# B&R Automation Studio project AAU12Segmenter (part 7)

#### DemoProgram.st - not listed in the package file held
```iecst
ACTION demoProgramTask:
	positionContainerDemo_0[0].initXPos := 0.060;
	positionContainerDemo_0[0].initYPos := 0.120;
	positionContainerDemo_0[1].initXPos := 0.180;
	positionContainerDemo_0[1].initYPos := 0.120;
	positionContainerDemo_0[2].initXPos := 0.300;
	positionContainerDemo_0[2].initYPos := 0.120;
	positionContainerDemo_0[3].initXPos := 0.420;
	positionContainerDemo_0[3].initYPos := 0.120;

	//Setup
	positionContainerLinkMovement[0].Shuttle3.xPos := 0.120;
	positionContainerLinkMovement[0].Shuttle3.yPos := 0.120;
	positionContainerLinkMovement[0].Shuttle2.xPos := 0.360;
	positionContainerLinkMovement[0].Shuttle2.yPos := 0.360;
	positionContainerLinkMovement[0].Shuttle4.xPos := 0.360;
	positionContainerLinkMovement[0].Shuttle4.yPos := 0.120;
	positionContainerLinkMovement[0].Shuttle1.xPos := 0.120;
	positionContainerLinkMovement[0].Shuttle1.yPos := 0.360;

	positionContainerLinkMovement[1].Shuttle3.xPos := 0.060;
	positionContainerLinkMovement[1].Shuttle3.yPos := 0.060;
	positionContainerLinkMovement[1].Shuttle2.xPos := 0.180;
	positionContainerLinkMovement[1].Shuttle2.yPos := 0.180;
	positionContainerLinkMovement[1].Shuttle4.xPos := 0.180;
	positionContainerLinkMovement[1].Shuttle4.yPos := 0.060;
	positionContainerLinkMovement[1].Shuttle1.xPos := 0.060;
	positionContainerLinkMovement[1].Shuttle1.yPos := 0.180;

	positionContainerLinkMovement[2].Shuttle3.xPos := 0.120;
	positionContainerLinkMovement[2].Shuttle3.yPos := 0.120;
	positionContainerLinkMovement[2].Shuttle2.xPos := 0.360;
	positionContainerLinkMovement[2].Shuttle2.yPos := 0.360;
	positionContainerLinkMovement[2].Shuttle4.xPos := 0.360;
	positionContainerLinkMovement[2].Shuttle4.yPos := 0.120;
	positionContainerLinkMovement[2].Shuttle1.xPos := 0.120;
	positionContainerLinkMovement[2].Shuttle1.yPos := 0.360;

	positionContainerLinkMovement[3].Shuttle3.xPos := 0.300;
	positionContainerLinkMovement[3].Shuttle3.yPos := 0.060;
	positionContainerLinkMovement[3].Shuttle2.xPos := 0.420;
	positionContainerLinkMovement[3].Shuttle2.yPos := 0.180;
	positionContainerLinkMovement[3].Shuttle4.xPos := 0.420;
	positionContainerLinkMovement[3].Shuttle4.yPos := 0.060;
	positionContainerLinkMovement[3].Shuttle1.xPos := 0.300;
	positionContainerLinkMovement[3].Shuttle1.yPos := 0.180;

	positionContainerLinkMovement[4].Shuttle3.xPos := 0.120;
	positionContainerLinkMovement[4].Shuttle3.yPos := 0.120;
	positionContainerLinkMovement[4].Shuttle2.xPos := 0.360;
	positionContainerLinkMovement[4].Shuttle2.yPos := 0.360;
	positionContainerLinkMovement[4].Shuttle4.xPos := 0.360;
	positionContainerLinkMovement[4].Shuttle4.yPos := 0.120;
	positionContainerLinkMovement[4].Shuttle1.xPos := 0.120;
	positionContainerLinkMovement[4].Shuttle1.yPos := 0.360;

	positionContainerLinkMovement[5].Shuttle3.xPos := 0.300;
	positionContainerLinkMovement[5].Shuttle3.yPos := 0.300;
	positionContainerLinkMovement[5].Shuttle2.xPos := 0.420;
	positionContainerLinkMovement[5].Shuttle2.yPos := 0.420;
	positionContainerLinkMovement[5].Shuttle4.xPos := 0.420;
	positionContainerLinkMovement[5].Shuttle4.yPos := 0.300;
	positionContainerLinkMovement[5].Shuttle1.xPos := 0.300;
	positionContainerLinkMovement[5].Shuttle1.yPos := 0.420;

	positionContainerLinkMovement[6].Shuttle3.xPos := 0.120;
	positionContainerLinkMovement[6].Shuttle3.yPos := 0.120;
	positionContainerLinkMovement[6].Shuttle2.xPos := 0.360;
	positionContainerLinkMovement[6].Shuttle2.yPos := 0.360;
	positionContainerLinkMovement[6].Shuttle4.xPos := 0.360;
	positionContainerLinkMovement[6].Shuttle4.yPos := 0.120;
	positionContainerLinkMovement[6].Shuttle1.xPos := 0.120;
	positionContainerLinkMovement[6].Shuttle1.yPos := 0.360;

	CASE em.substate OF
		5000:

			em.description := 'Move shuttle to pre pos';
			tempShuttleCounter := 0;
			MC_BR_MoveInPlaneAsync_Acp6D_0.Parameters.Acceleration := gAcp6DCtrl.Par.Acceleration;
			MC_BR_MoveInPlaneAsync_Acp6D_0.Parameters.Velocity := gAcp6DCtrl.Par.Velocity;
			FOR i := 0 TO UINT_TO_USINT(localCurrentNumShuttles-1) DO
				MC_BR_MoveInPlaneAsync_Acp6D_0.Parameters.AsyncPar[i].Shuttle := ADR(gAcp6DCtrl.Status.ShuttleInfo[i].shuttleRef);
				MC_BR_MoveInPlaneAsync_Acp6D_0.Parameters.AsyncPar[i].X := positionContainerDemo_0[i].initXPos;
				MC_BR_MoveInPlaneAsync_Acp6D_0.Parameters.AsyncPar[i].Y := positionContainerDemo_0[i].initYPos;
			END_FOR
			MC_BR_MoveInPlaneAsync_Acp6D_0.Execute := TRUE;
			IF MC_BR_MoveInPlaneAsync_Acp6D_0.Acknowledge THEN
				MC_BR_MoveInPlaneAsync_Acp6D_0.Execute := FALSE;
				em.substate := 5010;
			END_IF

		5010:
			MC_BR_MacroRun_Acp6D_0.Name := 'shuttleWave';
			MC_BR_MacroRun_Acp6D_0.Shuttle := ADR(gAcp6DCtrl.Status.ShuttleInfo[0].shuttleRef);
			MC_BR_MacroRun_Acp6D_0.Execute := TRUE;
			IF MC_BR_MacroRun_Acp6D_0.Acknowledge THEN
				MC_BR_MacroRun_Acp6D_0.Execute := FALSE;
				em.substate := 5015;
			END_IF

		5015:
			TON_0.PT := t#500ms;
			TON_0.IN := TRUE;
			IF TON_0.Q THEN
				TON_0.IN := FALSE;
				em.substate := 5020;
			END_IF

		5020:
			MC_BR_MacroRun_Acp6D_0.Name := 'shuttleWave';
			MC_BR_MacroRun_Acp6D_0.Shuttle := ADR(gAcp6DCtrl.Status.ShuttleInfo[1].shuttleRef);
			MC_BR_MacroRun_Acp6D_0.Execute := TRUE;
			IF MC_BR_MacroRun_Acp6D_0.Acknowledge THEN
				MC_BR_MacroRun_Acp6D_0.Execute := FALSE;
				em.substate := 5025;
			END_IF

		5025:
			TON_0.PT := t#500ms;
			TON_0.IN := TRUE;
			IF TON_0.Q THEN
				TON_0.IN := FALSE;
				em.substate := 5030;
			END_IF

		5030:
			MC_BR_MacroRun_Acp6D_0.Name := 'shuttleWave';
			MC_BR_MacroRun_Acp6D_0.Shuttle := ADR(gAcp6DCtrl.Status.ShuttleInfo[2].shuttleRef);
			MC_BR_MacroRun_Acp6D_0.Execute := TRUE;
			IF MC_BR_MacroRun_Acp6D_0.Acknowledge THEN
				MC_BR_MacroRun_Acp6D_0.Execute := FALSE;
				em.substate := 5035;
			END_IF

		5035:
			TON_0.PT := t#500ms;
			TON_0.IN := TRUE;
			IF TON_0.Q THEN
				TON_0.IN := FALSE;
				em.substate := 5040;
			END_IF

		5040:
			MC_BR_MacroRun_Acp6D_0.Name := 'shuttleWave';
			MC_BR_MacroRun_Acp6D_0.Shuttle := ADR(gAcp6DCtrl.Status.ShuttleInfo[3].shuttleRef);
			MC_BR_MacroRun_Acp6D_0.Execute := TRUE;
			IF MC_BR_MacroRun_Acp6D_0.Acknowledge THEN
				MC_BR_MacroRun_Acp6D_0.Execute := FALSE;
				em.substate := 5045;
			END_IF

		5045:
			em.description := 'Check all shuttle state';
			IF gAcp6DCtrl.Status.ShuttleInfo[0].State = mcACP6D_SH_STATE_IDLING AND gAcp6DCtrl.Status.ShuttleInfo[1].State = mcACP6D_SH_STATE_IDLING
				AND gAcp6DCtrl.Status.ShuttleInfo[2].State = mcACP6D_SH_STATE_IDLING AND gAcp6DCtrl.Status.ShuttleInfo[3].State = mcACP6D_SH_STATE_IDLING AND MC_BR_AsmReadStatus_Acp6D_0.AssemblyReady THEN
				em.substate := 5050;
			END_IF

		5050:
			em.description := 'Couple ShuttleGroup1_2';
			em.cmd.sc := FALSE;
			MC_BR_ShGroupCoupleCtrl_Acp6D_0.ShuttleGroup := shGroupShuttle1_2;
			MC_BR_ShGroupCoupleCtrl_Acp6D_0.Parameters.Option := 1; //Couple
			MC_BR_ShGroupCoupleCtrl_Acp6D_0.Execute := TRUE;
			IF MC_BR_ShGroupCoupleCtrl_Acp6D_0.Done THEN
				MC_BR_ShGroupCoupleCtrl_Acp6D_0.Execute := FALSE;
				em.substate := 5060;
			END_IF

		5060:
			em.description := 'Couple ShuttleGroup3_4';
			em.cmd.sc := FALSE;
			MC_BR_ShGroupCoupleCtrl_Acp6D_0.ShuttleGroup := shGroupShuttle3_4;
			MC_BR_ShGroupCoupleCtrl_Acp6D_0.Parameters.Option := 1; //Couple
			MC_BR_ShGroupCoupleCtrl_Acp6D_0.Execute := TRUE;
			IF MC_BR_ShGroupCoupleCtrl_Acp6D_0.Done THEN
				MC_BR_ShGroupCoupleCtrl_Acp6D_0.Execute := FALSE;
				em.substate := 5070;
			END_IF

		5070:
			em.cmd.sc := FALSE;
			MC_BR_MoveInPlane_Acp6D_0.Shuttle := ADR(gAcp6DCtrl.Status.ShuttleInfo[0].shuttleRef);
			MC_BR_MoveInPlane_Acp6D_0.Parameters.Position.X := 0.060;
			MC_BR_MoveInPlane_Acp6D_0.Parameters.Position.Y := 0.060;
			MC_BR_MoveInPlane_Acp6D_0.Parameters.Velocity := gAcp6DCtrl.Par.Velocity;
			MC_BR_MoveInPlane_Acp6D_0.Parameters.Acceleration := gAcp6DCtrl.Par.Acceleration;
			MC_BR_MoveInPlane_Acp6D_0.Parameters.Mode := 0; //Abs
			MC_BR_MoveInPlane_Acp6D_0.Parameters.Path := 0; //direct
			MC_BR_MoveInPlane_Acp6D_0.Execute := TRUE;
			IF MC_BR_MoveInPlane_Acp6D_0.Acknowledge THEN
				MC_BR_MoveInPlane_Acp6D_0.Execute := FALSE;
				em.substate := 5080;
			END_IF

		5080:
			em.cmd.sc := FALSE;
			MC_BR_MoveInPlane_Acp6D_0.Shuttle := ADR(gAcp6DCtrl.Status.ShuttleInfo[0].shuttleRef);
			MC_BR_MoveInPlane_Acp6D_0.Parameters.Position.X := 0.300;
			MC_BR_MoveInPlane_Acp6D_0.Parameters.Position.Y := 0.060;
			MC_BR_MoveInPlane_Acp6D_0.Parameters.Velocity := gAcp6DCtrl.Par.Velocity;
			MC_BR_MoveInPlane_Acp6D_0.Parameters.Acceleration := gAcp6DCtrl.Par.Acceleration;
			MC_BR_MoveInPlane_Acp6D_0.Parameters.Mode := 0; //Abs
			MC_BR_MoveInPlane_Acp6D_0.Parameters.Path := 0; //direct
			MC_BR_MoveInPlane_Acp6D_0.Execute := TRUE;
			IF MC_BR_MoveInPlane_Acp6D_0.Acknowledge THEN
				MC_BR_MoveInPlane_Acp6D_0.Execute := FALSE;
				em.substate := 5090;
			END_IF

		5090:
			em.cmd.sc := FALSE;
			MC_BR_MoveInPlane_Acp6D_0.Shuttle := ADR(gAcp6DCtrl.Status.ShuttleInfo[0].shuttleRef);
			MC_BR_MoveInPlane_Acp6D_0.Parameters.Position.X := 0.060;
			MC_BR_MoveInPlane_Acp6D_0.Parameters.Position.Y := 0.060;
			MC_BR_MoveInPlane_Acp6D_0.Parameters.Velocity := gAcp6DCtrl.Par.Velocity;
			MC_BR_MoveInPlane_Acp6D_0.Parameters.Acceleration := gAcp6DCtrl.Par.Acceleration;
			MC_BR_MoveInPlane_Acp6D_0.Parameters.Mode := 0; //Abs
			MC_BR_MoveInPlane_Acp6D_0.Parameters.Path := 0; //direct
			MC_BR_MoveInPlane_Acp6D_0.Execute := TRUE;
			IF MC_BR_MoveInPlane_Acp6D_0.Acknowledge THEN
				MC_BR_MoveInPlane_Acp6D_0.Execute := FALSE;
				em.substate := 5100;
			END_IF

		5100:
			em.cmd.sc := FALSE;
			MC_BR_MoveInPlane_Acp6D_0.Shuttle := ADR(gAcp6DCtrl.Status.ShuttleInfo[0].shuttleRef);
			MC_BR_MoveInPlane_Acp6D_0.Parameters.Position.X := 0.300;
			MC_BR_MoveInPlane_Acp6D_0.Parameters.Position.Y := 0.060;
			MC_BR_MoveInPlane_Acp6D_0.Parameters.Velocity := gAcp6DCtrl.Par.Velocity;
			MC_BR_MoveInPlane_Acp6D_0.Parameters.Acceleration := gAcp6DCtrl.Par.Acceleration;
			MC_BR_MoveInPlane_Acp6D_0.Parameters.Mode := 0; //Abs
			MC_BR_MoveInPlane_Acp6D_0.Parameters.Path := 0; //direct
			MC_BR_MoveInPlane_Acp6D_0.Execute := TRUE;
			IF MC_BR_MoveInPlane_Acp6D_0.Acknowledge THEN
				MC_BR_MoveInPlane_Acp6D_0.Execute := FALSE;
				em.substate := 5110;
			END_IF

		5110:
			em.cmd.sc := FALSE;
			MC_BR_MoveInPlane_Acp6D_0.Shuttle := ADR(gAcp6DCtrl.Status.ShuttleInfo[0].shuttleRef);
			MC_BR_MoveInPlane_Acp6D_0.Parameters.Position.X := 0.060;
			MC_BR_MoveInPlane_Acp6D_0.Parameters.Position.Y := 0.060;
			MC_BR_MoveInPlane_Acp6D_0.Parameters.Velocity := gAcp6DCtrl.Par.Velocity;
			MC_BR_MoveInPlane_Acp6D_0.Parameters.Acceleration := gAcp6DCtrl.Par.Acceleration;
			MC_BR_MoveInPlane_Acp6D_0.Parameters.Mode := 0; //Abs
			MC_BR_MoveInPlane_Acp6D_0.Parameters.Path := 0; //direct
			MC_BR_MoveInPlane_Acp6D_0.Execute := TRUE;
			IF MC_BR_MoveInPlane_Acp6D_0.Acknowledge THEN
				MC_BR_MoveInPlane_Acp6D_0.Execute := FALSE;
				em.substate := 5120;
			END_IF

		5120:
			em.cmd.sc := FALSE;
			MC_BR_MoveInPlane_Acp6D_0.Shuttle := ADR(gAcp6DCtrl.Status.ShuttleInfo[0].shuttleRef);
			MC_BR_MoveInPlane_Acp6D_0.Parameters.Position.X := 0.300;
			MC_BR_MoveInPlane_Acp6D_0.Parameters.Position.Y := 0.060;
			MC_BR_MoveInPlane_Acp6D_0.Parameters.Velocity := gAcp6DCtrl.Par.Velocity;
			MC_BR_MoveInPlane_Acp6D_0.Parameters.Acceleration := gAcp6DCtrl.Par.Acceleration;
			MC_BR_MoveInPlane_Acp6D_0.Parameters.Mode := 0; //Abs
			MC_BR_MoveInPlane_Acp6D_0.Parameters.Path := 0; //direct
			MC_BR_MoveInPlane_Acp6D_0.Execute := TRUE;
			IF MC_BR_MoveInPlane_Acp6D_0.Acknowledge THEN
				MC_BR_MoveInPlane_Acp6D_0.Execute := FALSE;
				em.substate := 5130;
			END_IF

		5130:
			em.cmd.sc := FALSE;
			MC_BR_MoveInPlane_Acp6D_0.Shuttle := ADR(gAcp6DCtrl.Status.ShuttleInfo[0].shuttleRef);
			MC_BR_MoveInPlane_Acp6D_0.Parameters.Position.X := 0.060;
			MC_BR_MoveInPlane_Acp6D_0.Parameters.Position.Y := 0.060;
			MC_BR_MoveInPlane_Acp6D_0.Parameters.Velocity := gAcp6DCtrl.Par.Velocity;
			MC_BR_MoveInPlane_Acp6D_0.Parameters.Acceleration := gAcp6DCtrl.Par.Acceleration;
			MC_BR_MoveInPlane_Acp6D_0.Parameters.Mode := 0; //Abs
			MC_BR_MoveInPlane_Acp6D_0.Parameters.Path := 0; //direct
			MC_BR_MoveInPlane_Acp6D_0.Execute := TRUE;
			IF MC_BR_MoveInPlane_Acp6D_0.Acknowledge THEN
				MC_BR_MoveInPlane_Acp6D_0.Execute := FALSE;
				em.substate := 5135;
			END_IF

		5135:
			em.cmd.sc := FALSE;
			MC_BR_MoveInPlane_Acp6D_0.Shuttle := ADR(gAcp6DCtrl.Status.ShuttleInfo[0].shuttleRef);
			MC_BR_MoveInPlane_Acp6D_0.Parameters.Position.X := 0.060;
			MC_BR_MoveInPlane_Acp6D_0.Parameters.Position.Y := 0.180;
			MC_BR_MoveInPlane_Acp6D_0.Parameters.Velocity := gAcp6DCtrl.Par.Velocity;
			MC_BR_MoveInPlane_Acp6D_0.Parameters.Acceleration := gAcp6DCtrl.Par.Acceleration;
			MC_BR_MoveInPlane_Acp6D_0.Parameters.Mode := 0; //Abs
			MC_BR_MoveInPlane_Acp6D_0.Parameters.Path := 0; //direct
			MC_BR_MoveInPlane_Acp6D_0.Execute := TRUE;
			IF MC_BR_MoveInPlane_Acp6D_0.Acknowledge THEN
				MC_BR_MoveInPlane_Acp6D_0.Execute := FALSE;
				em.substate := 5140;
			END_IF

		5140:
			em.cmd.sc := FALSE;
			MC_BR_MoveInPlane_Acp6D_0.Shuttle := ADR(gAcp6DCtrl.Status.ShuttleInfo[2].shuttleRef);
			MC_BR_MoveInPlane_Acp6D_0.Parameters.Position.X := 0.060;
			MC_BR_MoveInPlane_Acp6D_0.Parameters.Position.Y := 0.180;
			MC_BR_MoveInPlane_Acp6D_0.Parameters.Velocity := gAcp6DCtrl.Par.Velocity;
			MC_BR_MoveInPlane_Acp6D_0.Parameters.Acceleration := gAcp6DCtrl.Par.Acceleration;
			MC_BR_MoveInPlane_Acp6D_0.Parameters.Mode := 0; //Abs
			MC_BR_MoveInPlane_Acp6D_0.Parameters.Path := 0; //direct
			MC_BR_MoveInPlane_Acp6D_0.Execute := TRUE;
			IF MC_BR_MoveInPlane_Acp6D_0.Acknowledge THEN
				MC_BR_MoveInPlane_Acp6D_0.Execute := FALSE;
				em.substate := 5150;
			END_IF

		5150:
			em.cmd.sc := FALSE;
			MC_BR_MoveInPlane_Acp6D_0.Shuttle := ADR(gAcp6DCtrl.Status.ShuttleInfo[2].shuttleRef);
			MC_BR_MoveInPlane_Acp6D_0.Parameters.Position.X := 0.300;
			MC_BR_MoveInPlane_Acp6D_0.Parameters.Position.Y := 0.180;
			MC_BR_MoveInPlane_Acp6D_0.Parameters.Velocity := gAcp6DCtrl.Par.Velocity;
			MC_BR_MoveInPlane_Acp6D_0.Parameters.Acceleration := gAcp6DCtrl.Par.Acceleration;
			MC_BR_MoveInPlane_Acp6D_0.Parameters.Mode := 0; //Abs
			MC_BR_MoveInPlane_Acp6D_0.Parameters.Path := 0; //direct
			MC_BR_MoveInPlane_Acp6D_0.Execute := TRUE;
			IF MC_BR_MoveInPlane_Acp6D_0.Acknowledge THEN
				MC_BR_MoveInPlane_Acp6D_0.Execute := FALSE;
				em.substate := 5160;
			END_IF

		5160:
			em.cmd.sc := FALSE;
			MC_BR_MoveInPlane_Acp6D_0.Shuttle := ADR(gAcp6DCtrl.Status.ShuttleInfo[2].shuttleRef);
			MC_BR_MoveInPlane_Acp6D_0.Parameters.Position.X := 0.060;
			MC_BR_MoveInPlane_Acp6D_0.Parameters.Position.Y := 0.180;
			MC_BR_MoveInPlane_Acp6D_0.Parameters.Velocity := gAcp6DCtrl.Par.Velocity;
			MC_BR_MoveInPlane_Acp6D_0.Parameters.Acceleration := gAcp6DCtrl.Par.Acceleration;
			MC_BR_MoveInPlane_Acp6D_0.Parameters.Mode := 0; //Abs
			MC_BR_MoveInPlane_Acp6D_0.Parameters.Path := 0; //direct
			MC_BR_MoveInPlane_Acp6D_0.Execute := TRUE;
			IF MC_BR_MoveInPlane_Acp6D_0.Acknowledge THEN
				MC_BR_MoveInPlane_Acp6D_0.Execute := FALSE;
				em.substate := 5170;
			END_IF

		5170:
			em.cmd.sc := FALSE;
			MC_BR_MoveInPlane_Acp6D_0.Shuttle := ADR(gAcp6DCtrl.Status.ShuttleInfo[2].shuttleRef);
			MC_BR_MoveInPlane_Acp6D_0.Parameters.Position.X := 0.300;
			MC_BR_MoveInPlane_Acp6D_0.Parameters.Position.Y := 0.180;
			MC_BR_MoveInPlane_Acp6D_0.Parameters.Velocity := gAcp6DCtrl.Par.Velocity;
			MC_BR_MoveInPlane_Acp6D_0.Parameters.Acceleration := gAcp6DCtrl.Par.Acceleration;
			MC_BR_MoveInPlane_Acp6D_0.Parameters.Mode := 0; //Abs
			MC_BR_MoveInPlane_Acp6D_0.Parameters.Path := 0; //direct
			MC_BR_MoveInPlane_Acp6D_0.Execute := TRUE;
			IF MC_BR_MoveInPlane_Acp6D_0.Acknowledge THEN
				MC_BR_MoveInPlane_Acp6D_0.Execute := FALSE;
				em.substate := 5190;
			END_IF

		5190:
			em.cmd.sc := FALSE;
			MC_BR_MoveInPlane_Acp6D_0.Shuttle := ADR(gAcp6DCtrl.Status.ShuttleInfo[2].shuttleRef);
			MC_BR_MoveInPlane_Acp6D_0.Parameters.Position.X := 0.060;
			MC_BR_MoveInPlane_Acp6D_0.Parameters.Position.Y := 0.180;
			MC_BR_MoveInPlane_Acp6D_0.Parameters.Velocity := gAcp6DCtrl.Par.Velocity;
			MC_BR_MoveInPlane_Acp6D_0.Parameters.Acceleration := gAcp6DCtrl.Par.Acceleration;
			MC_BR_MoveInPlane_Acp6D_0.Parameters.Mode := 0; //Abs
			MC_BR_MoveInPlane_Acp6D_0.Parameters.Path := 0; //direct
			MC_BR_MoveInPlane_Acp6D_0.Execute := TRUE;
			IF MC_BR_MoveInPlane_Acp6D_0.Acknowledge THEN
				MC_BR_MoveInPlane_Acp6D_0.Execute := FALSE;
				em.substate := 5195;
			END_IF

		5195:
			em.cmd.sc := FALSE;
			MC_BR_MoveInPlane_Acp6D_0.Shuttle := ADR(gAcp6DCtrl.Status.ShuttleInfo[2].shuttleRef);
			MC_BR_MoveInPlane_Acp6D_0.Parameters.Position.X := 0.300;
			MC_BR_MoveInPlane_Acp6D_0.Parameters.Position.Y := 0.180;
			MC_BR_MoveInPlane_Acp6D_0.Parameters.Velocity := gAcp6DCtrl.Par.Velocity;
			MC_BR_MoveInPlane_Acp6D_0.Parameters.Acceleration := gAcp6DCtrl.Par.Acceleration;
			MC_BR_MoveInPlane_Acp6D_0.Parameters.Mode := 0; //Abs
			MC_BR_MoveInPlane_Acp6D_0.Parameters.Path := 0; //direct
			MC_BR_MoveInPlane_Acp6D_0.Execute := TRUE;
			IF MC_BR_MoveInPlane_Acp6D_0.Acknowledge THEN
				MC_BR_MoveInPlane_Acp6D_0.Execute := FALSE;
				em.substate := 5200;
			END_IF

		5200:
			em.description := 'DeCouple ShuttleGroup1_2';
			em.cmd.sc := FALSE;
			MC_BR_ShGroupCoupleCtrl_Acp6D_0.ShuttleGroup := shGroupShuttle1_2;
			MC_BR_ShGroupCoupleCtrl_Acp6D_0.Parameters.Option := 0; //DeCouple
			MC_BR_ShGroupCoupleCtrl_Acp6D_0.Execute := TRUE;
			IF MC_BR_ShGroupCoupleCtrl_Acp6D_0.Done THEN
				MC_BR_ShGroupCoupleCtrl_Acp6D_0.Execute := FALSE;
				em.substate := 5210;
			END_IF

		5210:
			em.description := 'DeCouple ShuttleGroup3_4';
			em.cmd.sc := FALSE;
			MC_BR_ShGroupCoupleCtrl_Acp6D_0.ShuttleGroup := shGroupShuttle3_4;
			MC_BR_ShGroupCoupleCtrl_Acp6D_0.Parameters.Option := 0; //DeCouple
			MC_BR_ShGroupCoupleCtrl_Acp6D_0.Execute := TRUE;
			IF MC_BR_ShGroupCoupleCtrl_Acp6D_0.Done THEN
				MC_BR_ShGroupCoupleCtrl_Acp6D_0.Execute := FALSE;
				em.substate := 5220;
			END_IF

		5220:
			em.description := 'check shuttle state idle';
			IF gAcp6DCtrl.Status.ShuttleInfo[0].State = mcACP6D_SH_STATE_IDLING AND gAcp6DCtrl.Status.ShuttleInfo[1].State = mcACP6D_SH_STATE_IDLING
				AND gAcp6DCtrl.Status.ShuttleInfo[2].State = mcACP6D_SH_STATE_IDLING AND gAcp6DCtrl.Status.ShuttleInfo[3].State = mcACP6D_SH_STATE_IDLING AND MC_BR_AsmReadStatus_Acp6D_0.AssemblyReady THEN
				em.substate := 5230;
			END_IF

		5230:
			em.description := 'Couple ShuttleGroup1_2';
			em.cmd.sc := FALSE;
			MC_BR_ShGroupCoupleCtrl_Acp6D_0.ShuttleGroup := shGroupShuttle1_2;
			MC_BR_ShGroupCoupleCtrl_Acp6D_0.Parameters.Option := 1; //Couple
			MC_BR_ShGroupCoupleCtrl_Acp6D_0.Execute := TRUE;
			IF MC_BR_ShGroupCoupleCtrl_Acp6D_0.Done THEN
				MC_BR_ShGroupCoupleCtrl_Acp6D_0.Execute := FALSE;
				em.substate := 5240;
			ELSIF MC_BR_ShGroupCoupleCtrl_Acp6D_0.Error THEN
				em.cmd.abort := TRUE;
			END_IF

		5240:
			em.description := 'Couple ShuttleGroup1_2';
			em.cmd.sc := FALSE;
			MC_BR_ShGroupCoupleCtrl_Acp6D_0.ShuttleGroup := shGroupShuttle3_4;
			MC_BR_ShGroupCoupleCtrl_Acp6D_0.Parameters.Option := 1; //Couple
			MC_BR_ShGroupCoupleCtrl_Acp6D_0.Execute := TRUE;
			IF MC_BR_ShGroupCoupleCtrl_Acp6D_0.Done THEN
				MC_BR_ShGroupCoupleCtrl_Acp6D_0.Execute := FALSE;
				em.substate := 5250;
			ELSIF MC_BR_ShGroupCoupleCtrl_Acp6D_0.Error THEN
				em.cmd.abort := TRUE;
			END_IF

		5250:
			em.description := 'Move group 10 of shuttle around';
			em.cmd.sc := FALSE;
			IF tempCounter >= 3 THEN
				tempCounter := 0;
				em.substate := 5270;
			ELSE
				MC_BR_MoveInPlane_Acp6D_0.Shuttle := ADR(gAcp6DCtrl.Status.ShuttleInfo[0].shuttleRef);
				MC_BR_MoveInPlane_Acp6D_0.Parameters.Position.X := 0.300;
				MC_BR_MoveInPlane_Acp6D_0.Parameters.Position.Y := 0.060;
				MC_BR_MoveInPlane_Acp6D_0.Parameters.Path := 2; //Y then X
				MC_BR_MoveInPlane_Acp6D_0.Execute := TRUE;
				IF MC_BR_MoveInPlane_Acp6D_0.Acknowledge THEN
					MC_BR_MoveInPlane_Acp6D_0.Execute := FALSE;
					em.substate := 5260;
				END_IF
			END_IF

		5260:
			em.description := 'Move group of shuttle around';
			em.cmd.sc := FALSE;
			MC_BR_MoveInPlane_Acp6D_0.Shuttle := ADR(gAcp6DCtrl.Status.ShuttleInfo[0].shuttleRef);
			MC_BR_MoveInPlane_Acp6D_0.Parameters.Position.X := 0.060;
			MC_BR_MoveInPlane_Acp6D_0.Parameters.Velocity := gAcp6DCtrl.Par.Velocity;
			MC_BR_MoveInPlane_Acp6D_0.Parameters.Acceleration := gAcp6DCtrl.Par.Acceleration;
			MC_BR_MoveInPlane_Acp6D_0.Parameters.Position.Y := 0.180;
			MC_BR_MoveInPlane_Acp6D_0.Parameters.Path := 2; //Y then X
			MC_BR_MoveInPlane_Acp6D_0.Execute := TRUE;
			IF MC_BR_MoveInPlane_Acp6D_0.Acknowledge THEN
				MC_BR_MoveInPlane_Acp6D_0.Execute := FALSE;
				tempCounter := tempCounter + 1;
				em.substate := 5250;
			END_IF

		5270:
			em.description := 'Move group 11 of shuttle around';
			em.cmd.sc := FALSE;
			IF tempCounter >= 3 THEN
				tempCounter := 0;
				em.substate := 5290;
			ELSE
				MC_BR_MoveInPlane_Acp6D_0.Shuttle := ADR(gAcp6DCtrl.Status.ShuttleInfo[2].shuttleRef);
				MC_BR_MoveInPlane_Acp6D_0.Parameters.Position.X := 0.060;
				MC_BR_MoveInPlane_Acp6D_0.Parameters.Position.Y := 0.180;
				MC_BR_MoveInPlane_Acp6D_0.Parameters.Path := 2; //Y then X
				MC_BR_MoveInPlane_Acp6D_0.Execute := TRUE;
				IF MC_BR_MoveInPlane_Acp6D_0.Acknowledge THEN
					MC_BR_MoveInPlane_Acp6D_0.Execute := FALSE;
					em.substate := 5280;
				END_IF
			END_IF

		5280:
			em.description := 'Move group of shuttle around';
			em.cmd.sc := FALSE;
			MC_BR_MoveInPlane_Acp6D_0.Shuttle := ADR(gAcp6DCtrl.Status.ShuttleInfo[2].shuttleRef);
			MC_BR_MoveInPlane_Acp6D_0.Parameters.Position.X := 0.300;
			MC_BR_MoveInPlane_Acp6D_0.Parameters.Velocity := gAcp6DCtrl.Par.Velocity;
			MC_BR_MoveInPlane_Acp6D_0.Parameters.Acceleration := gAcp6DCtrl.Par.Acceleration;
			MC_BR_MoveInPlane_Acp6D_0.Parameters.Position.Y := 0.060;
			MC_BR_MoveInPlane_Acp6D_0.Parameters.Path := 2; //Y then X
			MC_BR_MoveInPlane_Acp6D_0.Execute := TRUE;
			IF MC_BR_MoveInPlane_Acp6D_0.Acknowledge THEN
				MC_BR_MoveInPlane_Acp6D_0.Execute := FALSE;
				tempCounter := tempCounter + 1;
				em.substate := 5270;
			END_IF

		5290:
			em.description := 'DeCouple ShuttleGroup1_2';
			em.cmd.sc := FALSE;
			MC_BR_ShGroupCoupleCtrl_Acp6D_0.ShuttleGroup := shGroupShuttle1_2;
			MC_BR_ShGroupCoupleCtrl_Acp6D_0.Parameters.Option := 0; //DeCouple
			MC_BR_ShGroupCoupleCtrl_Acp6D_0.Execute := TRUE;
			IF MC_BR_ShGroupCoupleCtrl_Acp6D_0.Done THEN
				MC_BR_ShGroupCoupleCtrl_Acp6D_0.Execute := FALSE;
				em.substate := 5300;
			ELSIF MC_BR_ShGroupCoupleCtrl_Acp6D_0.Error THEN
				em.cmd.abort := TRUE;
			END_IF

		5300:
			em.description := 'Wait for shuttle to reach pos';
			em.cmd.sc := FALSE;
			IF((gAcp6DCtrl.Status.ShuttleInfo[2].Position.X > 0.300 - MARGIN AND gAcp6DCtrl.Status.ShuttleInfo[2].Position.X < 0.300 + MARGIN) AND
				gAcp6DCtrl.Status.ShuttleInfo[2].Position.Y > 0.060 - MARGIN AND gAcp6DCtrl.Status.ShuttleInfo[2].Position.Y < 0.060 + MARGIN) THEN
				IF gAcp6DCtrl.Status.ShuttleInfo[2].State = mcACP6D_SH_STATE_IDLING THEN
					em.substate := 5310;
				END_IF
			END_IF

		5310:
			em.description := 'Move right group up';
			em.cmd.sc := FALSE;
			MC_BR_MoveInPlane_Acp6D_0.Shuttle := ADR(gAcp6DCtrl.Status.ShuttleInfo[2].shuttleRef);
			MC_BR_MoveInPlane_Acp6D_0.Parameters.Position.X := 0.300;
			MC_BR_MoveInPlane_Acp6D_0.Parameters.Velocity := gAcp6DCtrl.Par.Velocity;
			MC_BR_MoveInPlane_Acp6D_0.Parameters.Acceleration := gAcp6DCtrl.Par.Acceleration;
			MC_BR_MoveInPlane_Acp6D_0.Parameters.Position.Y := 0.180;
			MC_BR_MoveInPlane_Acp6D_0.Parameters.Path := 0; //Direct
			MC_BR_MoveInPlane_Acp6D_0.Execute := TRUE;
			IF MC_BR_MoveInPlane_Acp6D_0.Acknowledge THEN
				MC_BR_MoveInPlane_Acp6D_0.Execute := FALSE;
				em.substate := 5320;
			END_IF

		5320:
			em.description := 'Couple ShuttleGroup1_2';
			em.cmd.sc := FALSE;
			MC_BR_ShGroupCoupleCtrl_Acp6D_0.ShuttleGroup := shGroupShuttle3_4;
			MC_BR_ShGroupCoupleCtrl_Acp6D_0.Parameters.Option := 0; //DeCouple
			MC_BR_ShGroupCoupleCtrl_Acp6D_0.Execute := TRUE;
			IF MC_BR_ShGroupCoupleCtrl_Acp6D_0.Done THEN
				MC_BR_ShGroupCoupleCtrl_Acp6D_0.Execute := FALSE;
				em.substate := 5330;
			ELSIF MC_BR_ShGroupCoupleCtrl_Acp6D_0.Error THEN
				em.cmd.abort := TRUE;
			END_IF

		5330:
			em.description := 'rotationMove part 1';
			MC_BR_MoveInPlane_Acp6D_0.Shuttle := ADR(gAcp6DCtrl.Status.ShuttleInfo[1].shuttleRef);
			MC_BR_MoveInPlane_Acp6D_0.Parameters.Position.X := 0.060;
			MC_BR_MoveInPlane_Acp6D_0.Parameters.Velocity := gAcp6DCtrl.Par.Velocity;
			MC_BR_MoveInPlane_Acp6D_0.Parameters.Acceleration := gAcp6DCtrl.Par.Acceleration;
			MC_BR_MoveInPlane_Acp6D_0.Parameters.Position.Y := 0.060;
			MC_BR_MoveInPlane_Acp6D_0.Parameters.Path := 2; //Y then X
			MC_BR_MoveInPlane_Acp6D_0.Execute := TRUE;
			IF MC_BR_MoveInPlane_Acp6D_0.Acknowledge THEN
				MC_BR_MoveInPlane_Acp6D_0.Execute := FALSE;
				em.substate := 5340;
			END_IF

		5340:
			em.description := 'rotationMove part 2';
			MC_BR_MoveInPlane_Acp6D_0.Shuttle := ADR(gAcp6DCtrl.Status.ShuttleInfo[3].shuttleRef);
			MC_BR_MoveInPlane_Acp6D_0.Parameters.Position.X := 0.180;
			MC_BR_MoveInPlane_Acp6D_0.Parameters.Velocity := gAcp6DCtrl.Par.Velocity;
			MC_BR_MoveInPlane_Acp6D_0.Parameters.Acceleration := gAcp6DCtrl.Par.Acceleration;
			MC_BR_MoveInPlane_Acp6D_0.Parameters.Position.Y := 0.060;
			MC_BR_MoveInPlane_Acp6D_0.Parameters.Path := 2; //Y then X
			MC_BR_MoveInPlane_Acp6D_0.Execute := TRUE;
			IF MC_BR_MoveInPlane_Acp6D_0.Acknowledge THEN
				MC_BR_MoveInPlane_Acp6D_0.Execute := FALSE;
				em.substate := 5350;
			END_IF

		5350:
			em.description := 'rotationMove part 3';
			MC_BR_MoveInPlane_Acp6D_0.Shuttle := ADR(gAcp6DCtrl.Status.ShuttleInfo[3].shuttleRef);
			MC_BR_MoveInPlane_Acp6D_0.Parameters.Position.X := 0.180;
			MC_BR_MoveInPlane_Acp6D_0.Parameters.Velocity := gAcp6DCtrl.Par.Velocity;
			MC_BR_MoveInPlane_Acp6D_0.Parameters.Acceleration := gAcp6DCtrl.Par.Acceleration;
			MC_BR_MoveInPlane_Acp6D_0.Parameters.Position.Y := 0.180;
			MC_BR_MoveInPlane_Acp6D_0.Parameters.Path := 0; //direct
			MC_BR_MoveInPlane_Acp6D_0.Execute := TRUE;
			IF MC_BR_MoveInPlane_Acp6D_0.Acknowledge THEN
				MC_BR_MoveInPlane_Acp6D_0.Execute := FALSE;
				em.substate := 5360;
			END_IF

		5360:
			em.description := 'Check switch is done part 1';
			IF((gAcp6DCtrl.Status.ShuttleInfo[3].Position.X > 0.180 - MARGIN AND gAcp6DCtrl.Status.ShuttleInfo[3].Position.X < 0.180 + MARGIN) AND
				gAcp6DCtrl.Status.ShuttleInfo[3].Position.Y > 0.180 - MARGIN AND gAcp6DCtrl.Status.ShuttleInfo[3].Position.Y < 0.180 + MARGIN) THEN
				IF gAcp6DCtrl.Status.ShuttleInfo[3].State = mcACP6D_SH_STATE_IDLING THEN
					em.substate := 5370;
				END_IF
			END_IF

		5370:
			em.description := 'rotationMove part 4';
			MC_BR_MoveInPlane_Acp6D_0.Shuttle := ADR(gAcp6DCtrl.Status.ShuttleInfo[1].shuttleRef);
			MC_BR_MoveInPlane_Acp6D_0.Parameters.Position.X := 0.420;
			MC_BR_MoveInPlane_Acp6D_0.Parameters.Velocity := gAcp6DCtrl.Par.Velocity;
			MC_BR_MoveInPlane_Acp6D_0.Parameters.Acceleration := gAcp6DCtrl.Par.Acceleration;
			MC_BR_MoveInPlane_Acp6D_0.Parameters.Position.Y := 0.180;
			MC_BR_MoveInPlane_Acp6D_0.Parameters.Path := 1; //X then Y
			MC_BR_MoveInPlane_Acp6D_0.Execute := TRUE;
			IF MC_BR_MoveInPlane_Acp6D_0.Acknowledge THEN
				MC_BR_MoveInPlane_Acp6D_0.Execute := FALSE;
				em.substate := 5380;
			END_IF

		5380:
			em.description := 'Check switch is done part 2';
			IF((gAcp6DCtrl.Status.ShuttleInfo[1].Position.X > 0.420 - MARGIN AND gAcp6DCtrl.Status.ShuttleInfo[1].Position.X < 0.420 + MARGIN) AND
				gAcp6DCtrl.Status.ShuttleInfo[1].Position.Y > 0.180 - MARGIN AND gAcp6DCtrl.Status.ShuttleInfo[1].Position.Y < 0.180 + MARGIN) THEN
				IF gAcp6DCtrl.Status.ShuttleInfo[1].State = mcACP6D_SH_STATE_IDLING THEN
					em.substate := 5390;
				END_IF
			END_IF

		5390:
			em.description := 'Couple ShuttleGroup1_4';
			em.cmd.sc := FALSE;
			MC_BR_ShGroupCoupleCtrl_Acp6D_0.ShuttleGroup := shGroupShuttle1_4;
			MC_BR_ShGroupCoupleCtrl_Acp6D_0.Parameters.Option := 1; //Couple
			MC_BR_ShGroupCoupleCtrl_Acp6D_0.Execute := TRUE;
			IF MC_BR_ShGroupCoupleCtrl_Acp6D_0.Done THEN
				MC_BR_ShGroupCoupleCtrl_Acp6D_0.Execute := FALSE;
				em.substate := 5400;
			ELSIF MC_BR_ShGroupCoupleCtrl_Acp6D_0.Error THEN
				em.cmd.abort := TRUE;
			END_IF

		5400:
			em.description := 'Couple ShuttleGroup2_3';
			em.cmd.sc := FALSE;
			MC_BR_ShGroupCoupleCtrl_Acp6D_0.ShuttleGroup := shGroupShuttle2_3;
			MC_BR_ShGroupCoupleCtrl_Acp6D_0.Parameters.Option := 1; //Couple
			MC_BR_ShGroupCoupleCtrl_Acp6D_0.Execute := TRUE;
			IF MC_BR_ShGroupCoupleCtrl_Acp6D_0.Done THEN
				MC_BR_ShGroupCoupleCtrl_Acp6D_0.Execute := FALSE;
				em.substate := 5410;
			ELSIF MC_BR_ShGroupCoupleCtrl_Acp6D_0.Error THEN
				em.cmd.abort := TRUE;
			END_IF

		5410:
			em.description := 'Move right side down';
			em.cmd.sc := FALSE;
			MC_BR_MoveInPlane_Acp6D_0.Shuttle := ADR(gAcp6DCtrl.Status.ShuttleInfo[2].shuttleRef);
			MC_BR_MoveInPlane_Acp6D_0.Parameters.Position.X := 0.300;
			MC_BR_MoveInPlane_Acp6D_0.Parameters.Velocity := gAcp6DCtrl.Par.Velocity;
			MC_BR_MoveInPlane_Acp6D_0.Parameters.Acceleration := gAcp6DCtrl.Par.Acceleration;
			MC_BR_MoveInPlane_Acp6D_0.Parameters.Position.Y := 0.060;
			MC_BR_MoveInPlane_Acp6D_0.Parameters.Path := 0; //direct
			MC_BR_MoveInPlane_Acp6D_0.Execute := TRUE;
			IF MC_BR_MoveInPlane_Acp6D_0.Acknowledge THEN
				MC_BR_MoveInPlane_Acp6D_0.Execute := FALSE;
				em.substate := 5430;
			END_IF

		5430:
			em.description := 'Move group 12 of shuttle around';
			em.cmd.sc := FALSE;
			IF tempCounter >= 3 THEN
				tempCounter := 0;
				em.substate := 5450;
			ELSE
				MC_BR_MoveInPlane_Acp6D_0.Shuttle := ADR(gAcp6DCtrl.Status.ShuttleInfo[0].shuttleRef);
				MC_BR_MoveInPlane_Acp6D_0.Parameters.Position.X := 0.300;
				MC_BR_MoveInPlane_Acp6D_0.Parameters.Position.Y := 0.060;
				MC_BR_MoveInPlane_Acp6D_0.Parameters.Path := 1; //X then Y
				MC_BR_MoveInPlane_Acp6D_0.Execute := TRUE;
				IF MC_BR_MoveInPlane_Acp6D_0.Acknowledge THEN
					MC_BR_MoveInPlane_Acp6D_0.Execute := FALSE;
					em.substate := 5440;
				END_IF
			END_IF

		5440:
			em.description := 'Move group of shuttle around';
			em.cmd.sc := FALSE;
			MC_BR_MoveInPlane_Acp6D_0.Shuttle := ADR(gAcp6DCtrl.Status.ShuttleInfo[0].shuttleRef);
			MC_BR_MoveInPlane_Acp6D_0.Parameters.Position.X := 0.060;
			MC_BR_MoveInPlane_Acp6D_0.Parameters.Velocity := gAcp6DCtrl.Par.Velocity;
			MC_BR_MoveInPlane_Acp6D_0.Parameters.Acceleration := gAcp6DCtrl.Par.Acceleration;
			MC_BR_MoveInPlane_Acp6D_0.Parameters.Position.Y := 0.180;
			MC_BR_MoveInPlane_Acp6D_0.Parameters.Path := 1; //X then Y
			MC_BR_MoveInPlane_Acp6D_0.Execute := TRUE;
			IF MC_BR_MoveInPlane_Acp6D_0.Acknowledge THEN
				MC_BR_MoveInPlane_Acp6D_0.Execute := FALSE;
				tempCounter := tempCounter + 1;
				em.substate := 5430;
			END_IF

		5450:
			em.description := 'Move group 13 of shuttle around';
			em.cmd.sc := FALSE;
			IF tempCounter >= 3 THEN
				tempCounter := 0;
				em.substate := 5470;
			ELSE
				MC_BR_MoveInPlane_Acp6D_0.Shuttle := ADR(gAcp6DCtrl.Status.ShuttleInfo[2].shuttleRef);
				MC_BR_MoveInPlane_Acp6D_0.Parameters.Position.X := 0.060;
				MC_BR_MoveInPlane_Acp6D_0.Parameters.Position.Y := 0.180;
				MC_BR_MoveInPlane_Acp6D_0.Parameters.Path := 1; //X then Y
				MC_BR_MoveInPlane_Acp6D_0.Execute := TRUE;
				IF MC_BR_MoveInPlane_Acp6D_0.Acknowledge THEN
					MC_BR_MoveInPlane_Acp6D_0.Execute := FALSE;
					em.substate := 5460;
				END_IF
			END_IF

		5460:
			em.description := 'Move group of shuttle around';
			em.cmd.sc := FALSE;
			MC_BR_MoveInPlane_Acp6D_0.Shuttle := ADR(gAcp6DCtrl.Status.ShuttleInfo[2].shuttleRef);
			MC_BR_MoveInPlane_Acp6D_0.Parameters.Position.X := 0.300;
			MC_BR_MoveInPlane_Acp6D_0.Parameters.Velocity := gAcp6DCtrl.Par.Velocity;
			MC_BR_MoveInPlane_Acp6D_0.Parameters.Acceleration := gAcp6DCtrl.Par.Acceleration;
			MC_BR_MoveInPlane_Acp6D_0.Parameters.Position.Y := 0.060;
			MC_BR_MoveInPlane_Acp6D_0.Parameters.Path := 1; //X then Y
			MC_BR_MoveInPlane_Acp6D_0.Execute := TRUE;
			IF MC_BR_MoveInPlane_Acp6D_0.Acknowledge THEN
				MC_BR_MoveInPlane_Acp6D_0.Execute := FALSE;
				tempCounter := tempCounter + 1;
				em.substate := 5450;
			END_IF

		5470:
			em.cmd.sc := FALSE;
			IF((gAcp6DCtrl.Status.ShuttleInfo[2].Position.X > 0.300 - MARGIN AND gAcp6DCtrl.Status.ShuttleInfo[2].Position.X < 0.300 + MARGIN) AND
				gAcp6DCtrl.Status.ShuttleInfo[2].Position.Y > 0.060 - MARGIN AND gAcp6DCtrl.Status.ShuttleInfo[2].Position.Y < 0.060 + MARGIN) THEN
				IF gAcp6DCtrl.Status.ShuttleInfo[2].State = mcACP6D_SH_STATE_IDLING THEN
					em.substate := 5480;
				END_IF
			END_IF

		5480:
			em.description := 'Move right group up';
			em.cmd.sc := FALSE;
			MC_BR_MoveInPlane_Acp6D_0.Shuttle := ADR(gAcp6DCtrl.Status.ShuttleInfo[2].shuttleRef);
			MC_BR_MoveInPlane_Acp6D_0.Parameters.Position.X := 0.300;
			MC_BR_MoveInPlane_Acp6D_0.Parameters.Velocity := gAcp6DCtrl.Par.Velocity;
			MC_BR_MoveInPlane_Acp6D_0.Parameters.Acceleration := gAcp6DCtrl.Par.Acceleration;
			MC_BR_MoveInPlane_Acp6D_0.Parameters.Position.Y := 0.180;
			MC_BR_MoveInPlane_Acp6D_0.Parameters.Path := 0; //Direct
			MC_BR_MoveInPlane_Acp6D_0.Execute := TRUE;
			IF MC_BR_MoveInPlane_Acp6D_0.Acknowledge THEN
				MC_BR_MoveInPlane_Acp6D_0.Execute := FALSE;
				em.substate := 5490;
			END_IF

		5490:
			em.description := 'DeCouple ShuttleGroup1_4';
			em.cmd.sc := FALSE;
			MC_BR_ShGroupCoupleCtrl_Acp6D_0.ShuttleGroup := shGroupShuttle1_4;
			MC_BR_ShGroupCoupleCtrl_Acp6D_0.Parameters.Option := 0; //DeCouple
			MC_BR_ShGroupCoupleCtrl_Acp6D_0.Execute := TRUE;
			IF MC_BR_ShGroupCoupleCtrl_Acp6D_0.Done THEN
				MC_BR_ShGroupCoupleCtrl_Acp6D_0.Execute := FALSE;
				em.substate := 5500;
			ELSIF MC_BR_ShGroupCoupleCtrl_Acp6D_0.Error THEN
				em.cmd.abort := TRUE;
			END_IF

		5500:
			em.description := 'DeCouple ShuttleGroup2_3';
			em.cmd.sc := FALSE;
			MC_BR_ShGroupCoupleCtrl_Acp6D_0.ShuttleGroup := shGroupShuttle2_3;
			MC_BR_ShGroupCoupleCtrl_Acp6D_0.Parameters.Option := 0; //DeCouple
			MC_BR_ShGroupCoupleCtrl_Acp6D_0.Execute := TRUE;
			IF MC_BR_ShGroupCoupleCtrl_Acp6D_0.Done THEN
				MC_BR_ShGroupCoupleCtrl_Acp6D_0.Execute := FALSE;
				em.substate := 5510;
			ELSIF MC_BR_ShGroupCoupleCtrl_Acp6D_0.Error THEN
				em.cmd.abort := TRUE;
			END_IF

		5510:
			em.description := 'rotationMove part 1';
			MC_BR_MoveInPlane_Acp6D_0.Shuttle := ADR(gAcp6DCtrl.Status.ShuttleInfo[3].shuttleRef);
			MC_BR_MoveInPlane_Acp6D_0.Parameters.Position.X := 0.060;
			MC_BR_MoveInPlane_Acp6D_0.Parameters.Velocity := gAcp6DCtrl.Par.Velocity;
			MC_BR_MoveInPlane_Acp6D_0.Parameters.Acceleration := gAcp6DCtrl.Par.Acceleration;
			MC_BR_MoveInPlane_Acp6D_0.Parameters.Position.Y := 0.060;
			MC_BR_MoveInPlane_Acp6D_0.Parameters.Path := 2; //Y then X
			MC_BR_MoveInPlane_Acp6D_0.Execute := TRUE;
			IF MC_BR_MoveInPlane_Acp6D_0.Acknowledge THEN
				MC_BR_MoveInPlane_Acp6D_0.Execute := FALSE;
				em.substate := 5520;
			END_IF

		5520:
			em.description := 'rotationMove part 2';
			MC_BR_MoveInPlane_Acp6D_0.Shuttle := ADR(gAcp6DCtrl.Status.ShuttleInfo[1].shuttleRef);
			MC_BR_MoveInPlane_Acp6D_0.Parameters.Position.X := 0.180;
			MC_BR_MoveInPlane_Acp6D_0.Parameters.Velocity := gAcp6DCtrl.Par.Velocity;
			MC_BR_MoveInPlane_Acp6D_0.Parameters.Acceleration := gAcp6DCtrl.Par.Acceleration;
			MC_BR_MoveInPlane_Acp6D_0.Parameters.Position.Y := 0.060;
			MC_BR_MoveInPlane_Acp6D_0.Parameters.Path := 2; //Y then X
			MC_BR_MoveInPlane_Acp6D_0.Execute := TRUE;
			IF MC_BR_MoveInPlane_Acp6D_0.Acknowledge THEN
				MC_BR_MoveInPlane_Acp6D_0.Execute := FALSE;
				em.substate := 5530;
			END_IF

		5530:
			em.description := 'rotationMove part 3';
			MC_BR_MoveInPlane_Acp6D_0.Shuttle := ADR(gAcp6DCtrl.Status.ShuttleInfo[1].shuttleRef);
			MC_BR_MoveInPlane_Acp6D_0.Parameters.Position.X := 0.180;
			MC_BR_MoveInPlane_Acp6D_0.Parameters.Velocity := gAcp6DCtrl.Par.Velocity;
			MC_BR_MoveInPlane_Acp6D_0.Parameters.Acceleration := gAcp6DCtrl.Par.Acceleration;
			MC_BR_MoveInPlane_Acp6D_0.Parameters.Position.Y := 0.180;
			MC_BR_MoveInPlane_Acp6D_0.Parameters.Path := 0; //direct
			MC_BR_MoveInPlane_Acp6D_0.Execute := TRUE;
			IF MC_BR_MoveInPlane_Acp6D_0.Acknowledge THEN
				MC_BR_MoveInPlane_Acp6D_0.Execute := FALSE;
				em.substate := 5540;
			END_IF

		5540:
			IF((gAcp6DCtrl.Status.ShuttleInfo[1].Position.X > 0.180 - MARGIN AND gAcp6DCtrl.Status.ShuttleInfo[1].Position.X < 0.180 + MARGIN) AND
				gAcp6DCtrl.Status.ShuttleInfo[1].Position.Y > 0.180 - MARGIN AND gAcp6DCtrl.Status.ShuttleInfo[1].Position.Y < 0.180 + MARGIN) THEN
				IF gAcp6DCtrl.Status.ShuttleInfo[1].State = mcACP6D_SH_STATE_IDLING THEN
					em.substate := 5550;
				END_IF
			END_IF

		5550:
			em.description := 'rotationMove part 4';
			MC_BR_MoveInPlane_Acp6D_0.Shuttle := ADR(gAcp6DCtrl.Status.ShuttleInfo[3].shuttleRef);
			MC_BR_MoveInPlane_Acp6D_0.Parameters.Position.X := 0.420;
			MC_BR_MoveInPlane_Acp6D_0.Parameters.Velocity := gAcp6DCtrl.Par.Velocity;
			MC_BR_MoveInPlane_Acp6D_0.Parameters.Acceleration := gAcp6DCtrl.Par.Acceleration;
			MC_BR_MoveInPlane_Acp6D_0.Parameters.Position.Y := 0.180;
			MC_BR_MoveInPlane_Acp6D_0.Parameters.Path := 1; //X then Y
			MC_BR_MoveInPlane_Acp6D_0.Execute := TRUE;
			IF MC_BR_MoveInPlane_Acp6D_0.Acknowledge THEN
				MC_BR_MoveInPlane_Acp6D_0.Execute := FALSE;
				em.substate := 5560;
			END_IF

		5560:
			IF((gAcp6DCtrl.Status.ShuttleInfo[3].Position.X > 0.420 - MARGIN AND gAcp6DCtrl.Status.ShuttleInfo[3].Position.X < 0.420 + MARGIN) AND
				gAcp6DCtrl.Status.ShuttleInfo[3].Position.Y > 0.180 - MARGIN AND gAcp6DCtrl.Status.ShuttleInfo[3].Position.Y < 0.180 + MARGIN) THEN
				IF gAcp6DCtrl.Status.ShuttleInfo[3].State = mcACP6D_SH_STATE_IDLING THEN
					em.substate := 5000;
				END_IF
			END_IF

//		5020:
//			em.description := 'Move shuttle up/down wave File 128-131';
//			MC_BR_MacroLoad_Acp6D_0.FileName := MC_BR_MacroList_Acp6D_0.MacroList[tempCounter];
//			MC_BR_MacroLoad_Acp6D_0.Execute := TRUE;
//			IF MC_BR_MacroLoad_Acp6D_0.Done THEN
//				tempCounter := tempCounter + 1;
//				MC_BR_MacroLoad_Acp6D_0.Execute := FALSE;
//				em.substate := 5021;
//			END_IF
//
//		5021:
//			em.description := 'check if all 4 shuttles have done wave move';
//			IF tempCounter > NUM_SHUTTLES THEN
//				em.substate := 5022;
//			ELSE
//				em.substate := 5020;
//			END_IF
//
//		5022:
//			em.description := 'Check shuttle 4 aka last shuttle reach pos';
//			IF((gAcp6DCtrl.Status.ShuttleInfo[3].Position.X > 0.420 - MARGIN AND gAcp6DCtrl.Status.ShuttleInfo[3].Position.X < 0.420 + MARGIN) AND
//				gAcp6DCtrl.Status.ShuttleInfo[3].Position.Y > 0.180 - MARGIN AND gAcp6DCtrl.Status.ShuttleInfo[3].Position.Y < 0.180 + MARGIN) THEN
//				IF gAcp6DCtrl.Status.ShuttleInfo[3].State = mcACP6D_SH_STATE_IDLING THEN
//					MC_BR_ZoneGetStatus_Acp6D_0.Execute := FALSE;
//					em.substate := 5030;
//				END_IF
//			END_IF
//
//		5030:
//			em.description := 'Link Shuttles';
//			em.description := 'Check if shuttle group 10 is created';
//			MC_BR_ShGroupGetStatus_Acp6D_0.GroupID := 10;
//			MC_BR_ShGroupGetStatus_Acp6D_0.Execute := TRUE;
//			IF MC_BR_ShGroupGetStatus_Acp6D_0.Done THEN
//				em.substate := 5031;
//			END_IF
//
//		5031:
//			IF MC_BR_ShGroupGetStatus_Acp6D_0.NumberOfShuttles > 0 THEN
//				//group created
//				MC_BR_ShGroupGetStatus_Acp6D_0.Execute := FALSE;
//				em.substate := 5032;
//			ELSE
//				//Create group
//				MC_BR_ShGroupGetStatus_Acp6D_0.Execute := FALSE;;
//				MC_BR_ShGroupCreate_Acp6D_0.GroupID := 10;
//				MC_BR_ShGroupCreate_Acp6D_0.NumberOfShuttles := 2;
//				MC_BR_ShGroupCreate_Acp6D_0.ShuttleID[0] := 1;
//				MC_BR_ShGroupCreate_Acp6D_0.ShuttleID[1] := 2;
//				//				MC_BR_ShGroupCreate_Acp6D_0.ShuttleID[2] := 3;
//				//				MC_BR_ShGroupCreate_Acp6D_0.ShuttleID[3] := 4;
//				MC_BR_ShGroupCreate_Acp6D_0.Execute := TRUE;
//				IF MC_BR_ShGroupCreate_Acp6D_0.Done THEN
//					MC_BR_ShGroupGetStatus_Acp6D_0.Execute := FALSE;
//					MC_BR_ShGroupCreate_Acp6D_0.Execute := FALSE;
//					em.substate := 5032;
//				END_IF
//			END_IF
//
//		5032:
//			em.description := 'Check if shuttle group 11 is created';
//			MC_BR_ShGroupGetStatus_Acp6D_0.GroupID := 11;
//			MC_BR_ShGroupGetStatus_Acp6D_0.Execute := TRUE;
//			IF MC_BR_ShGroupGetStatus_Acp6D_0.Done THEN
//				em.substate := 5033;
//			END_IF
//
//		5033:
//			IF MC_BR_ShGroupGetStatus_Acp6D_0.NumberOfShuttles > 0 THEN
//				//group created
//				MC_BR_ShGroupGetStatus_Acp6D_0.Execute := FALSE;
//				em.substate := 5040;
//			ELSE
//				//Create group
//				MC_BR_ShGroupGetStatus_Acp6D_0.Execute := FALSE;;
//				MC_BR_ShGroupCreate_Acp6D_0.GroupID := 11;
//				MC_BR_ShGroupCreate_Acp6D_0.NumberOfShuttles := 2;
//				MC_BR_ShGroupCreate_Acp6D_0.ShuttleID[0] := 3;
//				MC_BR_ShGroupCreate_Acp6D_0.ShuttleID[1] := 4;
//				//				MC_BR_ShGroupCreate_Acp6D_0.ShuttleID[2] := 3;
//				//				MC_BR_ShGroupCreate_Acp6D_0.ShuttleID[3] := 4;
//				MC_BR_ShGroupCreate_Acp6D_0.Execute := TRUE;
//				IF MC_BR_ShGroupCreate_Acp6D_0.Done THEN
//					MC_BR_ShGroupGetStatus_Acp6D_0.Execute := FALSE;
//					MC_BR_ShGroupCreate_Acp6D_0.Execute := FALSE;
//					em.substate := 5040;
//				END_IF
//			END_IF
//
//		5040:
//			em.description := 'couple shuttles group 10';
//			MC_BR_ShGroupCoupleCtrl_Acp6D_0.GroupID := 10;
//			MC_BR_ShGroupCoupleCtrl_Acp6D_0.CoupleMode := 0;
//			MC_BR_ShGroupCoupleCtrl_Acp6D_0.Option := 1; //Couple
//			MC_BR_ShGroupCoupleCtrl_Acp6D_0.Execute := TRUE;
//			IF MC_BR_ShGroupCoupleCtrl_Acp6D_0.Done THEN
//				MC_BR_ShGroupCoupleCtrl_Acp6D_0.Execute := FALSE;
//				em.substate := 5045;
//			END_IF
//
//		5045:
//			em.description := 'couple shuttles group 11';
//			MC_BR_ShGroupCoupleCtrl_Acp6D_0.GroupID := 11;
//			MC_BR_ShGroupCoupleCtrl_Acp6D_0.CoupleMode := 0;
//			MC_BR_ShGroupCoupleCtrl_Acp6D_0.Option := 1; //Couple
//			MC_BR_ShGroupCoupleCtrl_Acp6D_0.Execute := TRUE;
//			IF MC_BR_ShGroupCoupleCtrl_Acp6D_0.Done THEN
//				MC_BR_ShGroupCoupleCtrl_Acp6D_0.Execute := FALSE;
//				em.substate := 5050;
//			END_IF
//
//		5050:
//			em.description := 'prepaire tiktak move';
//			MC_BR_MoveInPlane_Acp6D_0.ShuttleID := 1;
//			MC_BR_MoveInPlane_Acp6D_0.PositionX := 0.060;
//			MC_BR_MoveInPlane_Acp6D_0.PositionY := 0.060;
//			MC_BR_MoveInPlane_Acp6D_0.Velocity := gAcp6DCtrl.Par.Velocity;
//			MC_BR_MoveInPlane_Acp6D_0.Acceleration := gAcp6DCtrl.Par.Acceleration;
//			MC_BR_MoveInPlane_Acp6D_0.Path := 2; //Y then X
//			MC_BR_MoveInPlane_Acp6D_0.Execute := TRUE;
//			IF MC_BR_MoveInPlane_Acp6D_0.Acknowledge THEN
//				MC_BR_MoveInPlane_Acp6D_0.Execute := FALSE;
//				em.substate := 5055;
//			END_IF
//
//		5055:
//			em.description := 'Move tiktak move File 132-135';
//			MC_BR_MacroLoad_Acp6D_0.FileName := MC_BR_MacroList_Acp6D_0.MacroList[tempCounter];
//			MC_BR_MacroLoad_Acp6D_0.Execute := TRUE;
//			IF MC_BR_MacroLoad_Acp6D_0.Done THEN
//				tempCounter := tempCounter + 1;
//				MC_BR_MacroLoad_Acp6D_0.Execute := FALSE;
//				em.substate := 5060;
//			END_IF
//
//		5060:
//			em.description := 'check if all 4 shuttles have done wave move';
//			IF tempCounter > 5 THEN
//				em.substate := 5065;
//			ELSE
//				em.substate := 5055;
//			END_IF
//
//		5065:
//			em.description := 'decouple shuttles group 10';
//			MC_BR_ShGroupCoupleCtrl_Acp6D_0.GroupID := 10;
//			MC_BR_ShGroupCoupleCtrl_Acp6D_0.CoupleMode := 0;
//			MC_BR_ShGroupCoupleCtrl_Acp6D_0.Option := 0; //Couple
//			MC_BR_ShGroupCoupleCtrl_Acp6D_0.Execute := TRUE;
//			IF MC_BR_ShGroupCoupleCtrl_Acp6D_0.Done THEN
//				MC_BR_ShGroupCoupleCtrl_Acp6D_0.Execute := FALSE;
//				em.substate := 5070;
//			END_IF
//
//		5070:
//			em.description := 'decouple shuttles group 11';
//			MC_BR_ShGroupCoupleCtrl_Acp6D_0.GroupID := 11;
//			MC_BR_ShGroupCoupleCtrl_Acp6D_0.CoupleMode := 0;
//			MC_BR_ShGroupCoupleCtrl_Acp6D_0.Option := 0; //Couple
//			MC_BR_ShGroupCoupleCtrl_Acp6D_0.Execute := TRUE;
//			IF MC_BR_ShGroupCoupleCtrl_Acp6D_0.Done THEN
//				MC_BR_ShGroupCoupleCtrl_Acp6D_0.Execute := FALSE;
//				em.substate := 5075;
//			END_IF
//
//		5075:
//			em.description := 'Move shuttle 3 to corner to make space for 2 shuttle show';
//			MC_BR_MoveInPlane_Acp6D_0.ShuttleID := 3;
//			MC_BR_MoveInPlane_Acp6D_0.PositionX := 0.420;
//			MC_BR_MoveInPlane_Acp6D_0.PositionY := 0.060;
//			MC_BR_MoveInPlane_Acp6D_0.Velocity := gAcp6DCtrl.Par.Velocity;
//			MC_BR_MoveInPlane_Acp6D_0.Acceleration := gAcp6DCtrl.Par.Acceleration;
//			MC_BR_MoveInPlane_Acp6D_0.Path := 2; //Y then X
//			MC_BR_MoveInPlane_Acp6D_0.Execute := TRUE;
//			IF MC_BR_MoveInPlane_Acp6D_0.Acknowledge THEN
//				MC_BR_MoveInPlane_Acp6D_0.Execute := FALSE;
//				em.substate := 5077;
//			END_IF
//
//		5077:
//			em.description := 'Check shuttle 3 reach pos';
//			IF((gAcp6DCtrl.Status.ShuttleInfo[2].Position.X > 0.420 - MARGIN AND gAcp6DCtrl.Status.ShuttleInfo[2].Position.X < 0.420 + MARGIN) AND
//				gAcp6DCtrl.Status.ShuttleInfo[2].Position.Y > 0.060 - MARGIN AND gAcp6DCtrl.Status.ShuttleInfo[2].Position.Y < 0.060 + MARGIN) THEN
//				IF gAcp6DCtrl.Status.ShuttleInfo[2].State = mcACP6D_SH_STATE_IDLING THEN
//					MC_BR_ZoneGetStatus_Acp6D_0.Execute := FALSE;
//					em.substate := 5080;
//				END_IF
//			END_IF
//
//		5080:
//			em.description := 'Move shuttle 2 a small amount away from shuttle 1';
//			MC_BR_MoveInPlane_Acp6D_0.ShuttleID := 2;
//			MC_BR_MoveInPlane_Acp6D_0.PositionX := 0.200;
//			MC_BR_MoveInPlane_Acp6D_0.PositionY := 0.060;
//			MC_BR_MoveInPlane_Acp6D_0.Velocity := gAcp6DCtrl.Par.Velocity;
//			MC_BR_MoveInPlane_Acp6D_0.Acceleration := gAcp6DCtrl.Par.Acceleration;
//			MC_BR_MoveInPlane_Acp6D_0.Path := 2; //Y then X
//			MC_BR_MoveInPlane_Acp6D_0.Execute := TRUE;
//			IF MC_BR_MoveInPlane_Acp6D_0.Done THEN
//				MC_BR_MoveInPlane_Acp6D_0.Execute := FALSE;
//				em.substate := 5085;
//			END_IF
//
//		5085:
//			em.description := 'couple shuttles group 10';
//			MC_BR_ShGroupCoupleCtrl_Acp6D_0.GroupID := 10;
//			MC_BR_ShGroupCoupleCtrl_Acp6D_0.CoupleMode := 0;
//			MC_BR_ShGroupCoupleCtrl_Acp6D_0.Option := 1; //Couple
//			MC_BR_ShGroupCoupleCtrl_Acp6D_0.Execute := TRUE;
//			IF MC_BR_ShGroupCoupleCtrl_Acp6D_0.Done THEN
//				MC_BR_ShGroupCoupleCtrl_Acp6D_0.Execute := FALSE;
//				em.substate := 5090;
//			END_IF
//
//		5090:
//			em.description := 'Move shuttles in X Y and RZ at the same time';
//			MC_BR_Move6D_Acp6D_0.Acceleration := 0.5;
//			MC_BR_Move6D_Acp6D_0.InPlaneVelocity := 0.14;
//			MC_BR_Move6D_Acp6D_0.ShuttleID := 1;
//			MC_BR_Move6D_Acp6D_0.ShortAxisVelocity[3] := 0.300;
//			MC_BR_Move6D_Acp6D_0.Position[0] := 0.140;
//			MC_BR_Move6D_Acp6D_0.Position[1] := 0.180;
//			MC_BR_Move6D_Acp6D_0.Position[2] := 0.001;
//			MC_BR_Move6D_Acp6D_0.Position[3] := 0;
//			MC_BR_Move6D_Acp6D_0.Position[4] := 0;
//			MC_BR_Move6D_Acp6D_0.Position[5] := 0.100;
//			MC_BR_Move6D_Acp6D_0.Execute := TRUE;
//			IF MC_BR_Move6D_Acp6D_0.Acknowledge THEN
//				MC_BR_Move6D_Acp6D_0.Execute := FALSE;
//				em.substate := 5095;
//			END_IF
//
//		5095:
//			em.description := 'Move shuttles in X Y and RZ at the same time';
//			MC_BR_Move6D_Acp6D_0.Acceleration := 0.5;
//			MC_BR_Move6D_Acp6D_0.InPlaneVelocity := 0.08;
//			MC_BR_Move6D_Acp6D_0.ShuttleID := 1;
//			MC_BR_Move6D_Acp6D_0.ShortAxisVelocity[3] := 0.300;
//			MC_BR_Move6D_Acp6D_0.Position[0] := 0.140;
//			MC_BR_Move6D_Acp6D_0.Position[1] := 0.060;
//			MC_BR_Move6D_Acp6D_0.Position[2] := 0.001;
//			MC_BR_Move6D_Acp6D_0.Position[3] := 0;
//			MC_BR_Move6D_Acp6D_0.Position[4] := 0;
//			MC_BR_Move6D_Acp6D_0.Position[5] := -0.100;
//			MC_BR_Move6D_Acp6D_0.Execute := TRUE;
//			IF MC_BR_Move6D_Acp6D_0.Acknowledge THEN
//				MC_BR_Move6D_Acp6D_0.Execute := FALSE;
//				em.substate := 5100;
//			END_IF
//
//		5100:
//			em.description := 'Move shuttles in X Y and RZ at the same time';
//			MC_BR_Move6D_Acp6D_0.Acceleration := 0.5;
//			MC_BR_Move6D_Acp6D_0.InPlaneVelocity := 0.1;
//			MC_BR_Move6D_Acp6D_0.ShuttleID := 1;
//			MC_BR_Move6D_Acp6D_0.ShortAxisVelocity[3] := 0.300;
//			MC_BR_Move6D_Acp6D_0.Position[0] := 0.060;
//			MC_BR_Move6D_Acp6D_0.Position[1] := 0.180;
//			MC_BR_Move6D_Acp6D_0.Position[2] := 0.001;
//			MC_BR_Move6D_Acp6D_0.Position[3] := 0;
//			MC_BR_Move6D_Acp6D_0.Position[4] := 0;
//			MC_BR_Move6D_Acp6D_0.Position[5] := 0.100;
//			MC_BR_Move6D_Acp6D_0.Execute := TRUE;
//			IF MC_BR_Move6D_Acp6D_0.Acknowledge THEN
//				MC_BR_Move6D_Acp6D_0.Execute := FALSE;
//				em.substate := 5105;
//			END_IF
//
//		5105:
//			em.description := 'Move shuttles in X Y and RZ at the same time';
//			MC_BR_Move6D_Acp6D_0.Acceleration := 0.5;
//			MC_BR_Move6D_Acp6D_0.InPlaneVelocity := 0.12;
//			MC_BR_Move6D_Acp6D_0.ShuttleID := 1;
//			MC_BR_Move6D_Acp6D_0.ShortAxisVelocity[3] := 0.300;
//			MC_BR_Move6D_Acp6D_0.Position[0] := 0.060;
//			MC_BR_Move6D_Acp6D_0.Position[1] := 0.060;
//			MC_BR_Move6D_Acp6D_0.Position[2] := 0.001;
//			MC_BR_Move6D_Acp6D_0.Position[3] := 0;
//			MC_BR_Move6D_Acp6D_0.Position[4] := 0;
//			MC_BR_Move6D_Acp6D_0.Position[5] := 0.0;
//			MC_BR_Move6D_Acp6D_0.Execute := TRUE;
//			IF MC_BR_Move6D_Acp6D_0.Acknowledge THEN
//				MC_BR_Move6D_Acp6D_0.Execute := FALSE;
//				IF tempCounter >= 8 THEN
//					tempCounter := 0;
//					em.substate := 5110;
//				ELSE
//					em.substate := 5090;
//					tempCounter := tempCounter + 1;
//				END_IF
//			END_IF
//
//		5110:
//			em.description := 'Decouple';
//			MC_BR_ShGroupCoupleCtrl_Acp6D_0.GroupID := 10;
//			MC_BR_ShGroupCoupleCtrl_Acp6D_0.CoupleMode := 0;
//			MC_BR_ShGroupCoupleCtrl_Acp6D_0.Option := 0; //Couple
//			MC_BR_ShGroupCoupleCtrl_Acp6D_0.Execute := TRUE;
//			IF MC_BR_ShGroupCoupleCtrl_Acp6D_0.Done THEN
//				MC_BR_ShGroupCoupleCtrl_Acp6D_0.Execute := FALSE;
//				em.substate := 5115;
//			END_IF
//
//		5115:
//			em.description := 'Check shuttle 1 reach pos';
//			IF((gAcp6DCtrl.Status.ShuttleInfo[0].Position.X > 0.060 - MARGIN AND gAcp6DCtrl.Status.ShuttleInfo[0].Position.X < 0.060 + MARGIN) AND
//				gAcp6DCtrl.Status.ShuttleInfo[0].Position.Y > 0.060 - MARGIN AND gAcp6DCtrl.Status.ShuttleInfo[0].Position.Y < 0.060 + MARGIN) THEN
//				IF gAcp6DCtrl.Status.ShuttleInfo[0].State = mcACP6D_SH_STATE_IDLING THEN
//					MC_BR_ZoneGetStatus_Acp6D_0.Execute := FALSE;
//					em.substate := 5010;
//				END_IF
//			END_IF
//
//
//
//
	END_CASE

	TON_0();

END_ACTION
```

#### KUKA.st - not listed in the package file held
```iecst
ACTION KUKA_program:

END_ACTION
```

#### MovementColumnSelection.st - not listed in the package file held
```iecst
FUNCTION_BLOCK MovementColumnSelection

	// Accessing the address
	availablePosition ACCESS ADR(availablePosition);

	// Determining the start and end row levels
	startRowLevel := PosToQuadrantIdx(pos := startWorkstation.par.departPosY);
	endRowLevel := PosToQuadrantIdx(pos := endWorkstation.par.approachPosY);

	// If the movementDone is not set, find the closest available column
	IF NOT opt_movementDone THEN
		FOR i := 0 TO 3 DO
			// Setting the index for the column looked at
			IF startWorkstation.par.workstationID <= 2 THEN
				selectedColumn := 3-i;
			ELSE
				selectedColumn := i;
			END_IF

			// Assume column is possible (and try to deny it)
			columnIsPossible := TRUE;

			// Going trough the rows the movement would go through and seing if it is possible
			FOR k := startRowLevel TO endRowLevel DO
				IF NOT availablePosition[selectedColumn, k] THEN
					columnIsPossible := FALSE;
					EXIT;
				END_IF
			END_FOR

			// If movement in the column is possible, occupy this column (selected column is already set)
			IF columnIsPossible THEN
				FOR k := startRowLevel TO endRowLevel DO
					availablePosition[selectedColumn, k] := FALSE;
				END_FOR
				EXIT;
			ELSE
				selectedColumn := -1;
			END_IF
		END_FOR
	ELSE
		FOR k := startRowLevel TO endRowLevel DO
			availablePosition[opt_resetColumn, k] := TRUE;
		END_FOR

		opt_resetColumn := FALSE;
		opt_movementDone := FALSE;
	END_IF

END_FUNCTION_BLOCK
```

#### ShuttleAtPosition.st - not listed in the package file held
```iecst
(* TODO: Add your comment here *)
FUNCTION_BLOCK ShuttleAtPosition

	IF (shuttlePos.X > checkPosX - MARGIN AND shuttlePos.X < checkPosX + MARGIN) AND
		(shuttlePos.Y > checkPosY - MARGIN AND shuttlePos.Y < checkPosY + MARGIN) THEN
		isAtCheckPos := TRUE;
	ELSE
		isAtCheckPos := FALSE;
	END_IF

END_FUNCTION_BLOCK
```

#### ShuttleIsAtPosition.st - not listed in the package file held
```iecst
(* TODO: Add your comment here *)
FUNCTION ShuttleIsAtPosition

	IF (shuttlePos.X > checkPosX - MARGIN AND shuttlePos.X < checkPosX + MARGIN) AND
		(shuttlePos.Y > checkPosY - MARGIN AND shuttlePos.Y < checkPosY + MARGIN) THEN
		ShuttleIsAtPosition := TRUE;
	ELSE
		ShuttleIsAtPosition := FALSE;
	END_IF

END_FUNCTION
```

#### SmartLab.st - not listed in the package file held
```iecst
ACTION smartLabWorkstationSetup:
	// Reset all workstations
	FOR i := 0 TO NR_OF_WORKSTATIONS DO
		gWorkStations[i].par.xLocation										:= 0.0;
		gWorkStations[i].par.yLocation										:= 0.0;
		gWorkStations[i].par.approachPosX									:= 0.0;
		gWorkStations[i].par.approachPosY									:= 0.0;
		gWorkStations[i].par.departPosX										:= 0.0;
		gWorkStations[i].par.departPosY										:= 0.0;
		gWorkStations[i].par.nextStationSelector							:= '0';
		gWorkStations[i].par.processTime									:= 0;
		gWorkStations[i].par.pathRouting									:= 0;
		gWorkStations[i].par.ArcMovement									:= FALSE;
		gWorkStations[i].par.landBeforeProcess								:= FALSE;
	END_FOR

	gWorkStations[0].par.xLocation										:= quadrantIdxToPos(5);
	gWorkStations[0].par.yLocation										:= quadrantIdxToPos(0);
	gWorkStations[0].par.approachPosX									:= quadrantIdxToPos(4);
	gWorkStations[0].par.approachPosY									:= quadrantIdxToPos(0);
	gWorkStations[0].par.departPosX										:= quadrantIdxToPos(4);
	gWorkStations[0].par.departPosY										:= quadrantIdxToPos(1);
	gWorkStations[0].par.nextStationSelector							:= '1';
	gWorkStations[0].par.processTime									:= 1.0;
	gWorkStations[0].par.pathRouting									:= 2; //Direct routing
	gWorkStations[0].par.ArcMovement									:= FALSE;
	gWorkStations[0].par.landBeforeProcess								:= FALSE;

	gWorkStations[1].par.xLocation										:= quadrantIdxToPos(5);
	gWorkStations[1].par.yLocation										:= quadrantIdxToPos(3);
	gWorkStations[1].par.approachPosX									:= quadrantIdxToPos(4);
	gWorkStations[1].par.approachPosY									:= quadrantIdxToPos(2);
	gWorkStations[1].par.departPosX										:= quadrantIdxToPos(4);
	gWorkStations[1].par.departPosY										:= quadrantIdxToPos(4);
	gWorkStations[1].par.nextStationSelector							:= '2';
	gWorkStations[1].par.processTime									:= 1.0;
	gWorkStations[1].par.pathRouting									:= 2;
	gWorkStations[1].par.ArcMovement									:= FALSE;
	gWorkStations[1].par.landBeforeProcess								:= FALSE;

	gWorkStations[2].par.xLocation										:= quadrantIdxToPos(5);
	gWorkStations[2].par.yLocation										:= quadrantIdxToPos(6);
	gWorkStations[2].par.approachPosX									:= quadrantIdxToPos(4);
	gWorkStations[2].par.approachPosY									:= quadrantIdxToPos(5);
	gWorkStations[2].par.departPosX										:= quadrantIdxToPos(4);
	gWorkStations[2].par.departPosY										:= quadrantIdxToPos(7);
	gWorkStations[2].par.nextStationSelector							:= '3';
	gWorkStations[2].par.processTime									:= 1.0;
	gWorkStations[2].par.pathRouting									:= 1;
	gWorkStations[2].par.ArcMovement									:= FALSE;
	gWorkStations[2].par.landBeforeProcess								:= FALSE;

	gWorkStations[3].par.xLocation										:= quadrantIdxToPos(0);
	gWorkStations[3].par.yLocation										:= quadrantIdxToPos(6);
	gWorkStations[3].par.approachPosX									:= quadrantIdxToPos(1);
	gWorkStations[3].par.approachPosY									:= quadrantIdxToPos(7);
	gWorkStations[3].par.departPosX										:= quadrantIdxToPos(1);
	gWorkStations[3].par.departPosY										:= quadrantIdxToPos(5);
	gWorkStations[3].par.nextStationSelector							:= '4';
	gWorkStations[3].par.processTime									:= 1.0;
	gWorkStations[3].par.pathRouting									:= 2;
	gWorkStations[3].par.ArcMovement									:= FALSE;
	gWorkStations[3].par.landBeforeProcess								:= FALSE;

	gWorkStations[4].par.xLocation										:= quadrantIdxToPos(0);
	gWorkStations[4].par.yLocation										:= quadrantIdxToPos(3);
	gWorkStations[4].par.approachPosX									:= quadrantIdxToPos(1);
	gWorkStations[4].par.approachPosY									:= quadrantIdxToPos(4);
	gWorkStations[4].par.departPosX										:= quadrantIdxToPos(1);
	gWorkStations[4].par.departPosY										:= quadrantIdxToPos(2);
	gWorkStations[4].par.nextStationSelector							:= '5';
	gWorkStations[4].par.processTime									:= 1.0;
	gWorkStations[4].par.pathRouting									:= 2;
	gWorkStations[4].par.ArcMovement									:= FALSE;
	gWorkStations[4].par.landBeforeProcess								:= TRUE;

	gWorkStations[5].par.xLocation										:= quadrantIdxToPos(0);
	gWorkStations[5].par.yLocation										:= quadrantIdxToPos(0);
	gWorkStations[5].par.approachPosX									:= quadrantIdxToPos(1);
	gWorkStations[5].par.approachPosY									:= quadrantIdxToPos(1);
	gWorkStations[5].par.departPosX										:= quadrantIdxToPos(1);
	gWorkStations[5].par.departPosY										:= quadrantIdxToPos(0);
	gWorkStations[5].par.nextStationSelector							:= '-1';
	gWorkStations[5].par.processTime									:= 1.0;
	gWorkStations[5].par.pathRouting									:= 1;
	gWorkStations[5].par.ArcMovement									:= FALSE;
	gWorkStations[5].par.landBeforeProcess								:= FALSE;

END_ACTION

ACTION smartLabSetup:

	positionContainerSmartLabProgram[0].initXPos := 0.420;
	positionContainerSmartLabProgram[0].initYPos := 0.300;

	positionContainerSmartLabProgram[2].initXPos := 0.420;
	positionContainerSmartLabProgram[2].initYPos := 0.420;

	positionContainerSmartLabProgram[4].initXPos := 0.420;
	positionContainerSmartLabProgram[4].initYPos := 0.540;

	positionContainerSmartLabProgram[6].initXPos := 0.420;
	positionContainerSmartLabProgram[6].initYPos := 0.660;

	positionContainerSmartLabProgram[1].initXPos := 0.300;
	positionContainerSmartLabProgram[1].initYPos := 0.300;

	positionContainerSmartLabProgram[3].initXPos := 0.300;
	positionContainerSmartLabProgram[3].initYPos := 0.420;

	positionContainerSmartLabProgram[5].initXPos := 0.300;
	positionContainerSmartLabProgram[5].initYPos := 0.540;

	positionContainerSmartLabProgram[7].initXPos := 0.300;
	positionContainerSmartLabProgram[7].initYPos := 0.660;

	smartLabWorkstationSetup; // Setup workstations

	FOR i := 0 TO NUM_SHUTTLES DO
		shuttleIndexAtPosition[i] := i;
		gShuttles[i].cm.state := 0;
		gWorkStations[i].cm.state := 0;
	END_FOR
	tempShuttleIndexAtPosition := shuttleIndexAtPosition;
	TON_0.IN := FALSE;
	bufferSize := SIZEOF(orderBuffer)/SIZEOF(orderBuffer[0]);

	CASE em.substate OF
		17000:
			em.description := 'Move shuttles to pre pos';
			MC_BR_MoveInPlaneAsync_Acp6D_0.Parameters.Acceleration := gAcp6DCtrl.Par.Acceleration;
			MC_BR_MoveInPlaneAsync_Acp6D_0.Parameters.Velocity := gAcp6DCtrl.Par.Velocity;
			FOR i := 0 TO UINT_TO_USINT(localCurrentNumShuttles-1) DO
				MC_BR_MoveInPlaneAsync_Acp6D_0.Parameters.AsyncPar[i].Shuttle := ADR(gAcp6DCtrl.Status.ShuttleInfo[i].shuttleRef);
				MC_BR_MoveInPlaneAsync_Acp6D_0.Parameters.AsyncPar[i].X := positionContainerSmartLabProgram[i].initXPos;
				MC_BR_MoveInPlaneAsync_Acp6D_0.Parameters.AsyncPar[i].Y := positionContainerSmartLabProgram[i].initYPos;
			END_FOR
			MC_BR_MoveInPlaneAsync_Acp6D_0.Execute := TRUE;
			IF MC_BR_MoveInPlaneAsync_Acp6D_0.Done THEN
				MC_BR_MoveInPlaneAsync_Acp6D_0.Execute := FALSE;
				em.substate := 17010;
			END_IF

	END_CASE
END_ACTION

ACTION smartLabInitialMovement:

	cm.description := 'Initiate movement to first workstation';
	IF moveToStartWorkstation[shuttleIndexAtPosition[i]] THEN
		pShuttle.function.MC_BR_MoveInPlane_Acp6D_0.Shuttle := ADR(gAcp6DCtrl.Status.ShuttleInfo[pShuttle.par.shuttleID].shuttleRef);
		pShuttle.function.MC_BR_MoveInPlane_Acp6D_0.Parameters.Acceleration := gAcp6DCtrl.Par.Acceleration;
		pShuttle.function.MC_BR_MoveInPlane_Acp6D_0.Parameters.Velocity := gAcp6DCtrl.Par.Velocity;
		pShuttle.function.MC_BR_MoveInPlane_Acp6D_0.Parameters.Position.X := gWorkStations[0].par.xLocation;
		pShuttle.function.MC_BR_MoveInPlane_Acp6D_0.Parameters.Position.Y := gWorkStations[0].par.yLocation;
		pShuttle.function.MC_BR_MoveInPlane_Acp6D_0.Parameters.Path := 2;
		pShuttle.function.MC_BR_MoveInPlane_Acp6D_0.Parameters.Mode := 0;

		pShuttle.function.MC_BR_MoveInPlane_Acp6D_0.Execute := TRUE;
		IF pShuttle.function.MC_BR_MoveInPlane_Acp6D_0.Acknowledge THEN
			pShuttle.function.MC_BR_MoveInPlane_Acp6D_0.Execute := FALSE;

			moveToStartWorkstation[shuttleIndexAtPosition[i]] := FALSE;
			//cm.state := 10;
		END_IF
	END_IF

	// Calls
	pShuttle.function.MC_BR_MoveInPlane_Acp6D_0();
	cm();

END_ACTION

ACTION smartLabWorkstationMovement:
	CASE cm.state OF
		0:
			cm.description := 'Check what shuttle is on top of workstation';
			FOR k := 0 TO (productOrder.amount - 1) DO
				IF (gAcp6DCtrl.Status.ShuttleInfo[shuttleIndexAtPosition[k]].Position.X > pWorkStations.par.xLocation - MARGIN AND gAcp6DCtrl.Status.ShuttleInfo[shuttleIndexAtPosition[k]].Position.X < pWorkStations.par.xLocation + MARGIN) AND
					(gAcp6DCtrl.Status.ShuttleInfo[shuttleIndexAtPosition[k]].Position.Y > pWorkStations.par.yLocation - MARGIN AND gAcp6DCtrl.Status.ShuttleInfo[shuttleIndexAtPosition[k]].Position.Y < pWorkStations.par.yLocation + MARGIN) THEN
					IF gAcp6DCtrl.Status.ShuttleInfo[shuttleIndexAtPosition[k]].State = mcACP6D_SH_STATE_IDLING THEN
						pWorkStations.par.tempShuttleID := shuttleIndexAtPosition[k];

						cm.state := 5;
					END_IF
				END_IF
			END_FOR

		5:
			cm.description := 'Send data to robot through mapping';
			CASE i OF
				0:
					orderSpec[0] := COVER_TYPE_TO_USINT(shuttlePlans[pWorkStations.par.tempShuttleID].productOrder.bottomCover);

				1:
					orderSpec[1] := shuttlePlans[pWorkStations.par.tempShuttleID].productOrder.Holes;

				2:
					orderSpec[2] := BOOL_TO_USINT(shuttlePlans[pWorkStations.par.tempShuttleID].productOrder.PCB);

				3:
					orderSpec[3] := shuttlePlans[pWorkStations.par.tempShuttleID].productOrder.Fuses;

				4:
					orderSpec[4] := COVER_TYPE_TO_USINT(shuttlePlans[pWorkStations.par.tempShuttleID].productOrder.topCover);

			END_CASE

			robotOperating[i] := TRUE; // Begin robot operation

			pWorkStations.TON_0.PT := REAL_TO_TIME(500); // Timer is needed for robot to start motion before shuttles moves away
			pWorkStations.TON_0.IN := TRUE;

			IF pWorkStations.TON_0.Q THEN
				pWorkStations.TON_0.IN := FALSE;
				IF pWorkStations.par.landBeforeProcess THEN
				cm.state := 10;
				ELSE
					cm.state := 20;
				END_IF
			END_IF

		10:
			cm.description := 'Land shuttle if required';
			IF gAcp6DCtrl.Status.ShuttleInfo[pWorkStations.par.tempShuttleID].State = mcACP6D_SH_STATE_IDLING THEN
				pWorkStations.MC_BR_ShLevitation_Acp6D_0.Shuttle := ADR(gAcp6DCtrl.Status.ShuttleInfo[pWorkStations.par.tempShuttleID].shuttleRef);
				pWorkStations.MC_BR_ShLevitation_Acp6D_0.Parameters.Level := 0; //Land
				pWorkStations.MC_BR_ShLevitation_Acp6D_0.Parameters.Speed := 0;
				pWorkStations.MC_BR_ShLevitation_Acp6D_0.Execute := TRUE;
			END_IF
			IF pWorkStations.MC_BR_ShLevitation_Acp6D_0.Done THEN
				pWorkStations.MC_BR_ShLevitation_Acp6D_0.Execute := FALSE;
				cm.state := 20;
			END_IF

		20:
			IF NOT robotOperating[i] THEN
				IF pWorkStations.par.landBeforeProcess THEN
					cm.state := 30;
				ELSE
					cm.state := 40;
				END_IF
			END_IF

		30:
			cm.description := 'Leviate shuttle if landed before process';
			pWorkStations.MC_BR_ShLevitation_Acp6D_0.Shuttle := ADR(gAcp6DCtrl.Status.ShuttleInfo[pWorkStations.par.tempShuttleID].shuttleRef);
			pWorkStations.MC_BR_ShLevitation_Acp6D_0.Parameters.Level := 1; //Leviate
			pWorkStations.MC_BR_ShLevitation_Acp6D_0.Parameters.Speed := 0;
			pWorkStations.MC_BR_ShLevitation_Acp6D_0.Execute := TRUE;
			IF pWorkStations.MC_BR_ShLevitation_Acp6D_0.Done THEN
				pWorkStations.MC_BR_ShLevitation_Acp6D_0.Execute := FALSE;
				cm.state := 40;
			END_IF

		40:
			cm.description := 'Move to next workstation';
			pWorkStations.MC_BR_MoveInPlane_Acp6D_0.Shuttle := ADR(gAcp6DCtrl.Status.ShuttleInfo[pWorkStations.par.tempShuttleID].shuttleRef);
			pWorkStations.MC_BR_MoveInPlane_Acp6D_0.Parameters.Velocity := gAcp6DCtrl.Par.Velocity;
			pWorkStations.MC_BR_MoveInPlane_Acp6D_0.Parameters.Acceleration := gAcp6DCtrl.Par.Acceleration;
			pWorkStations.MC_BR_MoveInPlane_Acp6D_0.Parameters.Mode := 0; //Absolute
			pWorkStations.MC_BR_MoveInPlane_Acp6D_0.Parameters.Path := pWorkStations.par.pathRouting; //0 Diagonal, 1 First X then Y, 2 First Y then X

			pTempShuttlePlan ACCESS ADR(shuttlePlans[pWorkStations.par.tempShuttleID]);
			pWorkStations.par.nextStationSelector := pTempShuttlePlan.routingSheet[pTempShuttlePlan.progressIndex];

			IF pWorkStations.par.nextStationSelector <> '-1' THEN
				pWorkStations.MC_BR_MoveInPlane_Acp6D_0.Parameters.Position.X := gWorkStations[STRING_TO_UDINT(pWorkStations.par.nextStationSelector)].par.xLocation;
				pWorkStations.MC_BR_MoveInPlane_Acp6D_0.Parameters.Position.Y := gWorkStations[STRING_TO_UDINT(pWorkStations.par.nextStationSelector)].par.yLocation;

				pWorkStations.MC_BR_MoveInPlane_Acp6D_0.Execute := TRUE;
				IF pWorkStations.MC_BR_MoveInPlane_Acp6D_0.Acknowledge THEN
					pWorkStations.MC_BR_MoveInPlane_Acp6D_0.Execute := FALSE;
					pTempShuttlePlan.progressIndex := pTempShuttlePlan.progressIndex + 1;
					cm.state := 0;
				END_IF
			ELSE
				pWorkStations.MC_BR_MoveInPlane_Acp6D_0.Parameters.Position.X := positionContainerSmartLabProgram[parkingSpotIndex].initXPos;
				pWorkStations.MC_BR_MoveInPlane_Acp6D_0.Parameters.Position.Y := positionContainerSmartLabProgram[parkingSpotIndex].initYPos;

				pWorkStations.MC_BR_MoveInPlane_Acp6D_0.Execute := TRUE;
				IF pWorkStations.MC_BR_MoveInPlane_Acp6D_0.Done THEN
					pWorkStations.MC_BR_MoveInPlane_Acp6D_0.Execute := FALSE;

					amountProductsFinished := amountProductsFinished + 1;
					tempShuttleIndexAtPosition[parkingSpotIndex] := pWorkStations.par.tempShuttleID; // Make the shuttle index correspond to the given position (see Smart Lab page for reference)
					parkingSpotIndex := parkingSpotIndex - 1;
					IF parkingSpotIndex = -1 THEN
						cm.state := 50;
					ELSE
						cm.state := 0;
					END_IF

				END_IF

			END_IF

		50:
			cm.description := 'Current product order has finished';
			orderFinished := TRUE;
			shuttleIndexAtPosition := tempShuttleIndexAtPosition;
			cm.state := 0;
			IF bufferEmpty THEN
				em.substate := 17010;
			ELSE
				em.substate := 17015;
			END_IF

	END_CASE

	//Calls
	pWorkStations.MC_BR_MoveInPlane_Acp6D_0();
	pWorkStations.MC_BR_MoveArc_Acp6D_0();
	pWorkStations.MC_BR_ShLevitation_Acp6D_0();
	pWorkStations.TON_0();
	cm();

END_ACTION
```

#### VisionMovement.st - not listed in the package file held
```iecst
ACTION VisionMovement:
	//Setup
//	MC_BR_ConfigReadCyclicCh_Acp6D_0.Controller := ADR(McAcp6DController);
//	FOR k := 0 TO NUM_SHUTTLES DO
//		MC_BR_ReadCyclicChAxis_Acp6D_0[0,k].Controller := ADR(McAcp6DController);
//		MC_BR_ReadCyclicChAxis_Acp6D_0[1,k].Controller := ADR(McAcp6DController);
//	END_FOR
//
	MC_BR_ReadCyclicPosition_Acp6D_0.Shuttle := ADR(gAcp6DCtrl.Status.ShuttleInfo[0].shuttleRef);
	//MC_BR_ReadCyclicPosition_Acp6D_0.Enable := TRUE;
	MC_BR_ReadCyclicPosition_Acp6D_1.Shuttle := ADR(gAcp6DCtrl.Status.ShuttleInfo[1].shuttleRef);
	//MC_BR_ReadCyclicPosition_Acp6D_1.Enable := TRUE;
	MC_BR_ReadCyclicPosition_Acp6D_2.Shuttle := ADR(gAcp6DCtrl.Status.ShuttleInfo[2].shuttleRef);
	//MC_BR_ReadCyclicPosition_Acp6D_2.Enable := TRUE;
	MC_BR_ReadCyclicPosition_Acp6D_3.Shuttle := ADR(gAcp6DCtrl.Status.ShuttleInfo[3].shuttleRef);
	//MC_BR_ReadCyclicPosition_Acp6D_3.Enable := TRUE;

	positionContainerVisionMovement[0].initXPos := 0.420;
	positionContainerVisionMovement[0].initYPos := 0.060;
	positionContainerVisionMovement[1].initXPos := 0.420;
	positionContainerVisionMovement[1].initYPos := 0.180;
	positionContainerVisionMovement[2].initXPos := 0.420;
	positionContainerVisionMovement[2].initYPos := 0.300;
	positionContainerVisionMovement[3].initXPos := 0.420;
	positionContainerVisionMovement[3].initYPos := 0.420;

	positionContainerVisionMovement[4].initXPos := 0.780;
	positionContainerVisionMovement[4].initYPos := 0.900;
	positionContainerVisionMovement[5].initXPos := 0.900;
	positionContainerVisionMovement[5].initYPos := 0.900;
	positionContainerVisionMovement[6].initXPos := 0.780;
	positionContainerVisionMovement[6].initYPos := 0.780;
	positionContainerVisionMovement[7].initXPos := 0.900;
	positionContainerVisionMovement[7].initYPos := 0.780;
	positionContainerVisionMovement[8].initXPos := 0.780;
	positionContainerVisionMovement[8].initYPos := 0.660;
	positionContainerVisionMovement[9].initXPos := 0.900;
	positionContainerVisionMovement[9].initYPos := 0.660;

	gWorkStations[0].par.xLocation										:= 0.000;
	gWorkStations[0].par.yLocation										:= 0.000;
	gWorkStations[0].par.nextStationSelector							:= '0';
	gWorkStations[0].par.processTime									:= 0;
	gWorkStations[0].par.pathRouting									:= 0;
	gWorkStations[0].par.ArcMovement									:= FALSE;

	gWorkStations[1].par.xLocation										:= 0.000;
	gWorkStations[1].par.yLocation										:= 0.000;
	gWorkStations[1].par.nextStationSelector							:= '0';
	gWorkStations[1].par.processTime									:= 0;
	gWorkStations[1].par.pathRouting									:= 0;
	gWorkStations[1].par.ArcMovement									:= FALSE;

	gWorkStations[2].par.xLocation										:= 0.060;
	gWorkStations[2].par.yLocation										:= 0.060;
	gWorkStations[2].par.nextStationSelector							:= '3';
	gWorkStations[2].par.processTime									:= 0;
	gWorkStations[2].par.pathRouting									:= 1;
	gWorkStations[2].par.ArcMovement									:= FALSE;

	gWorkStations[3].par.xLocation										:= 0.420;
	gWorkStations[3].par.yLocation										:= 0.420;
	gWorkStations[3].par.nextStationSelector							:= '2';
	gWorkStations[3].par.processTime									:= 3;
	gWorkStations[3].par.pathRouting									:= 1;
	gWorkStations[3].par.ArcMovement									:= FALSE;

	//visionLightControl
	IF controlLight.visionProgram THEN
		visionLightTON.PT := t#10s;
		visionLightTON.IN := TRUE;
		IF visionLightTON.Q THEN
			IF visionFlipFlop THEN
				visionFlipFlop := FALSE;
			ELSE
				visionFlipFlop := TRUE;
			END_IF
			visionLightTON.IN := FALSE;
		END_IF
		IF visionFlipFlop THEN
			lightValue := 1;
		ELSE
			lightValue := 8;
		END_IF
	END_IF

	CASE em.substate OF
		1000:
			em.description := 'Move shuttle to pre pos';
			MC_BR_MoveInPlaneAsync_Acp6D_0.Parameters.Acceleration := gAcp6DCtrl.Par.Acceleration;
			MC_BR_MoveInPlaneAsync_Acp6D_0.Parameters.Velocity := gAcp6DCtrl.Par.Velocity;
			FOR i := 0 TO UINT_TO_USINT(localCurrentNumShuttles-1) DO
				MC_BR_MoveInPlaneAsync_Acp6D_0.Parameters.AsyncPar[i].Shuttle := ADR(gAcp6DCtrl.Status.ShuttleInfo[i].shuttleRef);
				MC_BR_MoveInPlaneAsync_Acp6D_0.Parameters.AsyncPar[i].X := positionContainerVisionMovement[i].initXPos;
				MC_BR_MoveInPlaneAsync_Acp6D_0.Parameters.AsyncPar[i].Y := positionContainerVisionMovement[i].initYPos;
			END_FOR
			MC_BR_MoveInPlaneAsync_Acp6D_0.Execute := TRUE;
			IF MC_BR_MoveInPlaneAsync_Acp6D_0.Done THEN
				MC_BR_MoveInPlaneAsync_Acp6D_0.Execute := FALSE;
				em.substate := 1010;
			END_IF

		1010:
			em.description := 'Move shuttles towards workstation 1';
			IF tempShuttleCounter > 3 THEN
				tempShuttleCounter := 0;
				em.substate := 1023;
			ELSE
				MC_BR_MoveInPlane_Acp6D_0.Parameters.Acceleration := gAcp6DCtrl.Par.Acceleration;
				MC_BR_MoveInPlane_Acp6D_0.Parameters.Velocity := gAcp6DCtrl.Par.Velocity;
				MC_BR_MoveInPlane_Acp6D_0.Shuttle := ADR(gAcp6DCtrl.Status.ShuttleInfo[tempShuttleCounter].shuttleRef);
				MC_BR_MoveInPlane_Acp6D_0.Parameters.Position.X := 0.420;
				MC_BR_MoveInPlane_Acp6D_0.Parameters.Position.Y := 0.420;
				MC_BR_MoveInPlane_Acp6D_0.Parameters.Path := 1; //first x then y
				MC_BR_MoveInPlane_Acp6D_0.Parameters.Mode := 0;
				MC_BR_MoveInPlane_Acp6D_0.Execute := TRUE;
				IF MC_BR_MoveInPlane_Acp6D_0.Acknowledge THEN
					MC_BR_MoveInPlane_Acp6D_0.Execute := FALSE;
					tempShuttleCounter := tempShuttleCounter + 1;
					em.substate := 1020;
				END_IF
			END_IF

		1020:
			em.description := 'DummyScan';
			em.substate := 1010;

		1021:
//			em.description := 'Setup Cyclic channel';
//			MC_BR_ConfigReadCyclicCh_Acp6D_0.NumberOfChannels := 8;
//			MC_BR_ConfigReadCyclicCh_Acp6D_0.ChannelID[0] := 1;
//			MC_BR_ConfigReadCyclicCh_Acp6D_0.ChannelID[1] := 2;
//			MC_BR_ConfigReadCyclicCh_Acp6D_0.ChannelID[2] := 3;
//			MC_BR_ConfigReadCyclicCh_Acp6D_0.ChannelID[3] := 4;
//			MC_BR_ConfigReadCyclicCh_Acp6D_0.ChannelID[4] := 5;
//			MC_BR_ConfigReadCyclicCh_Acp6D_0.ChannelID[5] := 6;
//			MC_BR_ConfigReadCyclicCh_Acp6D_0.ChannelID[6] := 7;
//			MC_BR_ConfigReadCyclicCh_Acp6D_0.ChannelID[7] := 8;
//
//			MC_BR_ConfigReadCyclicCh_Acp6D_0.ShuttleID[0] := 1;
//			MC_BR_ConfigReadCyclicCh_Acp6D_0.ShuttleID[1] := 2;
//			MC_BR_ConfigReadCyclicCh_Acp6D_0.ShuttleID[2] := 3;
//			MC_BR_ConfigReadCyclicCh_Acp6D_0.ShuttleID[3] := 4;
//			MC_BR_ConfigReadCyclicCh_Acp6D_0.ShuttleID[4] := 1;
//			MC_BR_ConfigReadCyclicCh_Acp6D_0.ShuttleID[5] := 2;
//			MC_BR_ConfigReadCyclicCh_Acp6D_0.ShuttleID[6] := 3;
//			MC_BR_ConfigReadCyclicCh_Acp6D_0.ShuttleID[7] := 4;
//
//			MC_BR_ConfigReadCyclicCh_Acp6D_0.FeedbackMode[0] := 0;
//			MC_BR_ConfigReadCyclicCh_Acp6D_0.FeedbackMode[1] := 0;
//			MC_BR_ConfigReadCyclicCh_Acp6D_0.FeedbackMode[2] := 0;
//			MC_BR_ConfigReadCyclicCh_Acp6D_0.FeedbackMode[3] := 0;
//			MC_BR_ConfigReadCyclicCh_Acp6D_0.FeedbackMode[4] := 0;
//			MC_BR_ConfigReadCyclicCh_Acp6D_0.FeedbackMode[5] := 0;
//			MC_BR_ConfigReadCyclicCh_Acp6D_0.FeedbackMode[6] := 0;
//			MC_BR_ConfigReadCyclicCh_Acp6D_0.FeedbackMode[7] := 0;
//
//			MC_BR_ConfigReadCyclicCh_Acp6D_0.Execute := TRUE;
//
//			IF MC_BR_ConfigReadCyclicCh_Acp6D_0.Done THEN
//				MC_BR_ConfigReadCyclicCh_Acp6D_0.Execute := FALSE;
//				tempCounter := 1;
//				em.substate := 1022;
//			END_IF

		1022:
			em.description := 'Turn on channelStreaming';
//			FOR k := 0 TO 1 DO
//				FOR j := 0 TO NUM_SHUTTLES DO
//					MC_BR_ReadCyclicChAxis_Acp6D_0[k,j].AxisID := k+1;
//					MC_BR_ReadCyclicChAxis_Acp6D_0[k,j].ChannelID := tempCounter;
//					MC_BR_ReadCyclicChAxis_Acp6D_0[k,j].Enable := TRUE;
//					tempCounter := tempCounter + 1;
//				END_FOR
//			END_FOR
//			tempCounter := 1;
//			em.substate := 1023;

		1023:
			em.description := 'Check if camera has self adjusted';
			IF gVisionSensor[3].DAT.Focus > 0 AND gVisionSensor[3].DAT.Exposure > 0 THEN
				em.substate := 1030;
			ELSE
				em.substate := 1024;
			END_IF

		1024:
			em.description := 'Move shuttle to under camera before self adjust';
			MC_BR_MoveInPlane_Acp6D_0.Parameters.Acceleration := gAcp6DCtrl.Par.Acceleration;
			MC_BR_MoveInPlane_Acp6D_0.Parameters.Velocity := gAcp6DCtrl.Par.Velocity;
			MC_BR_MoveInPlane_Acp6D_0.Shuttle := ADR(gAcp6DCtrl.Status.ShuttleInfo[3].shuttleRef);
			MC_BR_MoveInPlane_Acp6D_0.Parameters.Position.X := 0.180;
			MC_BR_MoveInPlane_Acp6D_0.Parameters.Position.Y := 0.420;
			MC_BR_MoveInPlane_Acp6D_0.Execute := TRUE;
			IF MC_BR_MoveInPlane_Acp6D_0.Acknowledge THEN
				MC_BR_MoveInPlane_Acp6D_0.Execute := FALSE;
				em.substate := 1025;
			END_IF

		1025:
			em.description := 'Check pos reached';
			IF((gAcp6DCtrl.Status.ShuttleInfo[3].Position.X > 0.180 - MARGIN AND gAcp6DCtrl.Status.ShuttleInfo[3].Position.X < 0.180 + MARGIN) AND
				(gAcp6DCtrl.Status.ShuttleInfo[3].Position.Y > 0.420 - MARGIN AND gAcp6DCtrl.Status.ShuttleInfo[3].Position.Y < 0.420 + MARGIN)) THEN
				IF gAcp6DCtrl.Status.ShuttleInfo[3].State = mcACP6D_SH_STATE_IDLING THEN
					em.substate := 1026;
				END_IF
			END_IF

		1026:
			em.description := 'Fire autoSetup';
			gVisionSensor[3].CMD.AutoSetupStartStop := TRUE;
			em.substate := 1027;

		1027:
			em.description := 'Check when self calibration is done';
			IF NOT gVisionSensor[3].CMD.AutoSetupStartStop AND gVisionSensor[3].DAT.Focus > 0 AND gVisionSensor[3].DAT.Exposure > 0 THEN
				gVisionSensor[3].DAT.Exposure := 100; // known best camera value
				em.substate := 1028;
			END_IF

		1028:
			em.description := 'Move caliShuttle back';
			MC_BR_MoveInPlane_Acp6D_0.Parameters.Acceleration := gAcp6DCtrl.Par.Acceleration;
			MC_BR_MoveInPlane_Acp6D_0.Parameters.Velocity := gAcp6DCtrl.Par.Velocity;
			MC_BR_MoveInPlane_Acp6D_0.Shuttle := ADR(gAcp6DCtrl.Status.ShuttleInfo[3].shuttleRef);
			MC_BR_MoveInPlane_Acp6D_0.Parameters.Position.X := 0.060;
			MC_BR_MoveInPlane_Acp6D_0.Parameters.Position.Y := 0.060;
			MC_BR_MoveInPlane_Acp6D_0.Parameters.Path := 1; //x then y
			MC_BR_MoveInPlane_Acp6D_0.Execute := TRUE;
			IF MC_BR_MoveInPlane_Acp6D_0.Acknowledge THEN
				MC_BR_MoveInPlane_Acp6D_0.Execute := FALSE;
				em.substate := 1030;
			END_IF

		1030:
			em.description := 'Move shuttle with workStationMovement task and count laps';

	END_CASE
	MC_BR_ReadCyclicPosition_Acp6D_0.Enable := FALSE;
	MC_BR_ReadCyclicPosition_Acp6D_1.Enable := FALSE;
	MC_BR_ReadCyclicPosition_Acp6D_2.Enable := FALSE;
	MC_BR_ReadCyclicPosition_Acp6D_3.Enable := FALSE;

	CASE shuttleToTakePictureOf OF
		0:
			ShuttleYPos_m := MC_BR_ReadCyclicPosition_Acp6D_0.CyclicPosition.X;
			MC_BR_ReadCyclicPosition_Acp6D_0.Enable := TRUE;
		1:
			ShuttleYPos_m := MC_BR_ReadCyclicPosition_Acp6D_1.CyclicPosition.X;
			MC_BR_ReadCyclicPosition_Acp6D_1.Enable := TRUE;
		2:
			ShuttleYPos_m := MC_BR_ReadCyclicPosition_Acp6D_2.CyclicPosition.X;
			MC_BR_ReadCyclicPosition_Acp6D_2.Enable := TRUE;
		3:
			ShuttleYPos_m := MC_BR_ReadCyclicPosition_Acp6D_3.CyclicPosition.X;
			MC_BR_ReadCyclicPosition_Acp6D_3.Enable := TRUE;
	END_CASE

	//ShuttleYPos_m := SEL(MC_BR_ReadCyclicChAxis_Acp6D_0[0,shuttleToTakePictureOf-1].Valid,0,MC_BR_ReadCyclicChAxis_Acp6D_0[0,shuttleToTakePictureOf-1].Value);

//	MC_BR_ConfigReadCyclicCh_Acp6D_0(Controller := ADR(McAcp6DController));

//	FOR k := 0 TO NUM_SHUTTLES DO
//		MC_BR_ReadCyclicChAxis_Acp6D_0[0,k](Controller := ADR(McAcp6DController));
//		MC_BR_ReadCyclicChAxis_Acp6D_0[1,k](Controller := ADR(McAcp6DController));
//	END_FOR

	visionLightTON();

END_ACTION
```

### Types.typ
```iecst
TYPE
	Acp6DCmdType : 	STRUCT
		PowerOn : BOOL;
		PowerOff : BOOL;
		ErrorReset : BOOL;
		Init : BOOL;
		StartProcess : BOOL;
		StopProcess : BOOL;
		Stop : BOOL;
		gameProgramDeleteShuttle : BOOL;
	END_STRUCT;
	Acp6DCtrlType : 	STRUCT
		Cmd : Acp6DCmdType;
		Status : Acp6DStatusType;
		Par : Acp6DParType;
	END_STRUCT;
	Acp6DParType : 	STRUCT
		Acceleration : REAL := 10;
		Velocity : REAL := 2;
		modeSelector : driveModes;
		rotationVelocity : REAL := 200;
		rotationAcceleration : REAL := 10;
	END_STRUCT;
	Acp6DStatusType : 	STRUCT
		Error : BOOL;
		ErrorID : DINT;
		Ready : BOOL;
		PowerOn : BOOL;
		ReadyToPowerOn : BOOL;
		ShuttleInfo : ARRAY[0..NUM_SHUTTLES]OF ShuttleInfoType;
		ShuttleInfoVis : ARRAY[0..NUM_SHUTTLES]OF ShuttleInfoType;
		currentNumShuttles : UINT;
	END_STRUCT;
	box_typ : 	STRUCT
		smallBox : BOOL;
		bottle : BOOL;
		bigBox : BOOL;
		LastTypeWasBox : BOOL;
	END_STRUCT;
	driveModes :
		(
		none := 0, (*bootup*)
		vision := 1,
		weight := 2,
		linkMovement := 3,
		gameProgram := 4,
		demoProgram := 5,
		shuttleToConveyor := 6,
		workstationMovement := 8,
		conveyorStationMovement := 9,
		dialGauge := 7,
		danfossMode := 10,
		sunMovement := 11,
		flaskProgram := 12,
		boxProgram := 13,
		rotationProgram := 14,
		steelSheet := 15,
		test := 16,
		smartLab := 17
		);
	ShuttleInfoType : 	STRUCT
		ID : UINT;
		State : McAcp6DShStateEnum;
		Force : McAcp6DShForceType;
		Position : McAcp6DShPositionType;
		inUse : BOOL; (*DryStation Bool*)
		lastgPath : DINT := 100;
		shuttleRef : Mc6DShuttleType;
	END_STRUCT;
	shuttleStartup_typ : 	STRUCT
		initYPos : REAL;
		initXPos : REAL;
		nextStationSelector : STRING[80] := '0';
		initZPos : REAL;
		initRxPos : REAL;
		initRyPos : REAL;
		initRzPos : REAL;
	END_STRUCT;
	workStation_cmd_typ : 	STRUCT
		dummy : USINT;
	END_STRUCT;
	workStation_par_typ : 	STRUCT
		landBeforeProcess : BOOL; (*TRUE = yes*)
		yLocation : REAL;
		xLocation : REAL;
		tempShuttleID : USINT;
		processTime : REAL;
		pathRouting : USINT := 0; (*0 Diagonal, 1 First X then Y, 2 First Y then X*)
		nextStationSelector : STRING[80];
		ArcMovement : BOOL;
		internalCounter : USINT;
		tempCounter : USINT;
	END_STRUCT;
	workStation_status_typ : 	STRUCT
		componentName : STRING[80];
		active : BOOL;
		oneshot : BOOL;
	END_STRUCT;
	workStation_typ : 	STRUCT
		par : workStation_par_typ;
		status : workStation_status_typ;
		cmd : workStation_cmd_typ;
		cm : brdkCM;
		MC_BR_RotaryMotionSpin_Acp6D_0 : MC_BR_RotaryMotionSpin_Acp6D;
		MC_BR_RotaryMotion_Acp6D_0 : MC_BR_RotaryMotion_Acp6D;
		MC_BR_MoveInPlane_Acp6D_0 : MC_BR_MoveInPlane_Acp6D;
		MC_BR_ShLevitation_Acp6D_0 : MC_BR_ShLevitation_Acp6D;
		TON_0 : TON;
		workstationSwitcher : BOOL;
		MC_BR_MoveArc_Acp6D_0 : MC_BR_MoveArc_Acp6D;
		MC_BR_Move6D_Acp6D_0 : MC_BR_Move6D_Acp6D;
	END_STRUCT;
END_TYPE
```

### Variables.var
```iecst
VAR
	cmdBoxProgram : box_typ;
	gAcp6DCtrl : Acp6DCtrlType;
END_VAR
VAR CONSTANT
	NR_OF_WORKSTATIONS : USINT := 9; (*10[0..9]*)
	NUM_SHUTTLES : USINT := 7; (*8[0..7]*)
END_VAR
(*Constants*)
VAR
	shuttleStartupInfo : ARRAY[0..NUM_SHUTTLES] OF shuttleStartup_typ;
	ShuttleYPos_m : LREAL;
END_VAR
```

### Program Logical/Modules/KUKA/CTRL (IEC)

#### Types.typ - Local data types
```iecst
TYPE
	KUKA : 	STRUCT
		cm : brdkCM;
		init : init_function;
		motion : motion_function;
		read : read_function;
		status : status;
		operationType : operation_type;
		gripperType : gripper_type;
		gripperAction : GripperAction;
		TON : TON;
	END_STRUCT;
	init_function : 	STRUCT
		KRC_ReadAxisGroup : KRC_ReadAxisGroup;
		KRC_Initialize : KRC_Initialize;
		KRC_Error : KRC_Error;
		KRC_AutomaticExternal : KRC_AutomaticExternal;
		KRC_AutoStart : KRC_AutoStart;
		KRC_SetOverride : KRC_SetOverride;
		KRC_Diag : KRC_Diag;
		KRC_WriteAxisGroup : KRC_WriteAxisGroup;
	END_STRUCT;
	motion_function : 	STRUCT
		KRC_MoveDirectAbsolute : KRC_MoveDirectAbsolute;
		KRC_MoveDirectRelative : KRC_MoveDirectRelative;
		KRC_MoveLinearAbsolute : KRC_MoveLinearAbsolute;
		KRC_MoveLinearRelative : KRC_MoveLinearRelative;
	END_STRUCT;
	read_function : 	STRUCT
		KRC_ReadActualPosition : KRC_ReadActualPosition;
		KRC_ReadActualAxisPosition : KRC_ReadActualAxisPosition;
	END_STRUCT;
	operation_type :
		(
		ASSEMBLY := 0,
		PROCESS := 1
		);
	gripper_type :
		(
		COVER_GRIPPER := 0,
		PCB_GRIPPER := 1,
		FUSE_GRIPPER := 2
		);
	status : 	STRUCT
		S_ : BOOL;
		I_ : BOOL;
		R_ : BOOL;
		EXT_ : BOOL;
		P_ : BOOL;
	END_STRUCT;
	gripper_action_type :
		(
		OPEN := 0,
		CLOSE := 1
		);
END_TYPE
```

#### Variables.var - Local variables
```iecst
(*AxisStructure*)
VAR
	AxisRef : AXIS_GROUP_REF_ARR; (*Axis Reference of the Robot*)
END_VAR
(*Variables for the Task*)
(*Instance of mxA-FB*)
VAR
	KRC_Abort_0 : KRC_Abort; (*Function Block to abort actual movement*)
	KRC_AutomaticExternal_0 : KRC_AutomaticExternal; (*Function Block to Enable the Movement from the PLC*)
	KRC_AutomaticExternal_1 : KRC_AutomaticExternal; (*Function Block to Enable the Movement from the PLC*)
	KRC_AutoStart_0 : KRC_AutoStart; (*Function Block for Autostarting the Starting Chain of a Robot*)
	KRC_AutoStart_1 : KRC_AutoStart; (*Function Block for Autostarting the Starting Chain of a Robot*)
	KRC_Diag_0 : KRC_Diag; (*Function Block for getting Diagnostic information*)
	KRC_Diag_1 : KRC_Diag; (*Function Block for getting Diagnostic information*)
	KRC_Error_0 : KRC_Error; (*Function Block gives back Error Status*)
	KRC_Error_1 : KRC_Error; (*Function Block gives back Error Status*)
	KRC_Initialize_0 : KRC_Initialize; (*Function Block to Initialize the Robot*)
	KRC_Initialize_1 : KRC_Initialize; (*Function Block to Initialize the Robot*)
	KRC_ReadActualAxisPosition_0 : KRC_ReadActualAxisPosition; (*Function Block returns actual Axis Position (A1-A6)*)
	KRC_ReadActualPosition_0 : KRC_ReadActualPosition; (*Function Block returns actual Axis Position (X-C)*)
	KRC_ReadAxisGroup_0 : KRC_ReadAxisGroup; (*Function Block to Read the AxisInformation*)
	KRC_SetOverride_0 : KRC_SetOverride; (*Function Block to Set the Override*)
	KRC_SetOverride_1 : KRC_SetOverride; (*Function Block to Set the Override*)
	KRC_WriteAxisGroup_0 : KRC_WriteAxisGroup; (*Function Block to Write on the OutputVariable for controlling the Robot*)
	mxa_ValuesToCOORDSYS_0 : mxa_ValuesToCOORDSYS; (*Function Block to set int values to the Coordsys*)
END_VAR
(*Variables for UDP-communication*)
VAR
	i : USINT; (*IndexVariable for ErrorMessages*)
	InputUDPString : STRING[255]; (*Variable with Message from KRC*)
	counterMsg : INT;
	WorkAroundCounter : INT;
	step_UDPConnect : INT; (*State-Variable for Errorhandling*)
	TextArray : ARRAY[0..15] OF STRING[255]; (*TextArray contains Messages from KRC*)
	pState : INT := 0;
	UdpOpen_0 : UdpOpen; (*FunctionBlock to Open Port*)
	UdpOpen_1 : UdpOpen; (*FunctionBlock to Open Port*)
	UdpRecv_0 : UdpRecv; (*FunctionBlock to Receive Message*)
	UdpSend_0 : UdpSend; (*FunctionBlock to Send Message*)
	MsgToKrc : STRING[17]; (*Contains the Message which is send to KRC for getting all Messages*)
	ReloadMsg : BOOL; (*Variable triggers the Sequence to get Messages*)
END_VAR
VAR CONSTANT
	STATE_DISPLAY : INT := 5; (*STATE to display the Message*)
	STATE_RECEIVE : INT := 3; (*STATE to receive a new Message*)
	STATE_OPEN : INT := 0; (*STATE for opening the Ports*)
	STATE_SEND : INT := 2; (*STATE for sending a request to KRC*)
	STATE_WAIT : INT := 1; (*STATE for Waiting to trigger a new Request*)
END_VAR
VAR
	TON_0 : TON;
END_VAR
(*HMI Status KRC*)
VAR
	Status_EXT : INT; (*Variable used to show correct color in Visualization for the EXT-Shape*)
	Status_I : INT; (*Variable used to show correct color in Visualization for the I-Shape*)
	Status_P : INT; (*Variable used to show correct color in Visualization for the P-Shape*)
	Status_R : INT; (*Variable used to show correct color in Visualization for the R-Shape*)
	Status_S : INT; (*Variable used to show correct color in Visualization for the S-Shape*)
END_VAR
(*Misc*)
VAR
	KRC_MoveLinearAbsolute_0 : KRC_MoveLinearAbsolute;
	coordSys : COORDSYS;
	toolCover : FRAME;
	endPOS : E6POS;
	KRC_WriteToolData_0 : KRC_WriteToolData;
END_VAR
```

#### mxA_Main.st - Cyclic code
```iecst
PROGRAM _CYCLIC

	/////////////////////////////////////////////////////
	// Logic to transform USINT (Input) to BYTE (FUBS) //
	/////////////////////////////////////////////////////
	FOR i:=0 TO 5 DO
		brsmemcpy(ADR(KRC_Input[i,0]),ADR(InputVariables[i,0]), 254);
	END_FOR

	/////////////////////////////////////////////////////
	// KRC_ReadAxisGroup has to be called at the Begin //
	// of the Cyclic Task to get all the Information   //
	// From the KRC from KUKA						   //
	/////////////////////////////////////////////////////

	KRC_ReadAxisGroup_0.KRC4_Input 			:= ADR(KRC_Input[0,0]);
	KRC_ReadAxisGroup_0.AxisGroupIdx 		:= 1;
	KRC_ReadAxisGroup_0.KRC_AxisGroupRefArr := ADR(AxisRef);

	KRC_ReadAxisGroup_0();

	//KRC_ReadAxisGroup_1.KRC4_Input 			:= ADR(KRC4_Input_1);
	//KRC_ReadAxisGroup_1.AxisGroupIdx 		:= 2;
	//KRC_ReadAxisGroup_1.KRC_AxisGroupRefArr := ADR(AxisRef);

	//KRC_ReadAxisGroup_1();

	/////////////////////////////////////////////////////
	// Call User functions                             //
	/////////////////////////////////////////////////////

	mxA_Start;
	//mxA_Motion;
	//mxA_JointMovement;
	mxA_LinearMovement;
	//mxA_ErrorMessage;

	// Function calls from Motion.fbd
	KRC_ReadActualAxisPosition_0.AxisGroupIdx 			:= HMI_AxisGroup;
	KRC_ReadActualAxisPosition_0.KRC_AxisGroupRefArr 	:= ADR(AxisRef);
	KRC_ReadActualAxisPosition_0();

	HMI_A1 												:= KRC_ReadActualAxisPosition_0.A1;
	HMI_A2 												:= KRC_ReadActualAxisPosition_0.A2;
	HMI_A3 												:= KRC_ReadActualAxisPosition_0.A3;
	HMI_A4 												:= KRC_ReadActualAxisPosition_0.A4;
	HMI_A5 												:= KRC_ReadActualAxisPosition_0.A5;
	HMI_A6 												:= KRC_ReadActualAxisPosition_0.A6;

	KRC_ReadActualPosition_0.AxisGroupIdx 				:= HMI_AxisGroup;
	KRC_ReadActualPosition_0.KRC_AxisGroupRefArr 		:= ADR(AxisRef);
	KRC_ReadActualPosition_0();

	HMI_X												:= KRC_ReadActualPosition_0.X;
	HMI_Y												:= KRC_ReadActualPosition_0.Y;
	HMI_Z												:= KRC_ReadActualPosition_0.Z;
	HMI_A												:= KRC_ReadActualPosition_0.A;
	HMI_B												:= KRC_ReadActualPosition_0.B;
	HMI_C												:= KRC_ReadActualPosition_0.C;

	KRC_Abort_0.AxisGroupIdx 							:= HMI_AxisGroup;
	KRC_Abort_0.KRC_AxisGroupRefArr						:= ADR(AxisRef);
	KRC_Abort_0.ExecuteCmd								:= HMI_ExeAbort;
	KRC_Abort_0();

	/////////////////////////////////////////////////////
	// FunctionBlock to write the Output on the Struct //
	/////////////////////////////////////////////////////

	KRC_WriteAxisGroup_0.AxisGroupIdx			:= 1;
	KRC_WriteAxisGroup_0.KRC_AxisGroupRefArr 	:= ADR(AxisRef);
	KRC_WriteAxisGroup_0.KRC4_Output 			:= ADR(KRC4_Output);

	KRC_WriteAxisGroup_0();

	//KRC_WriteAxisGroup_1.AxisGroupIdx 			:= 2;
	//KRC_WriteAxisGroup_1.KRC_AxisGroupRefArr 	:= ADR(AxisRef);
	//KRC_WriteAxisGroup_1.KRC4_Output 			:= ADR(KRC4_Output_1);

	//KRC_WriteAxisGroup_1();

	/////////////////////////////////////////////////////
	// Logic to transform BYTE (FUBS) to USINT (Input) //
	/////////////////////////////////////////////////////
	FOR i:=0 TO 5 DO
		brsmemcpy(ADR(OutputVariables[i,0]),ADR(KRC_Output[i,0]), 254);
	END_FOR

	END_PROGRAM
```
